// LS Electric XG5000 project: LOADER ITMV X3353 SYSTEM 20250323
// PLC LSPLC
// module base 0 slot 1: Internal Analog Input/Output:XBF-AH08E (A/D Voltage/Current 4 Ch, D/A Voltage/Current 4 Ch)
// module base 0 slot 2: Positioning Module:XBF-PN04B (Position Control, EtherCAT Network Type(4 axis))
// module base 0 slot 3: Input Module:XBE-DC32A (DC 24V Input, 32 Contacts (Current Source Sink Input/Current Source Input))

PROGRAM MAIN (task: ½ºÄµ ÇÁ·Î±×·¥)

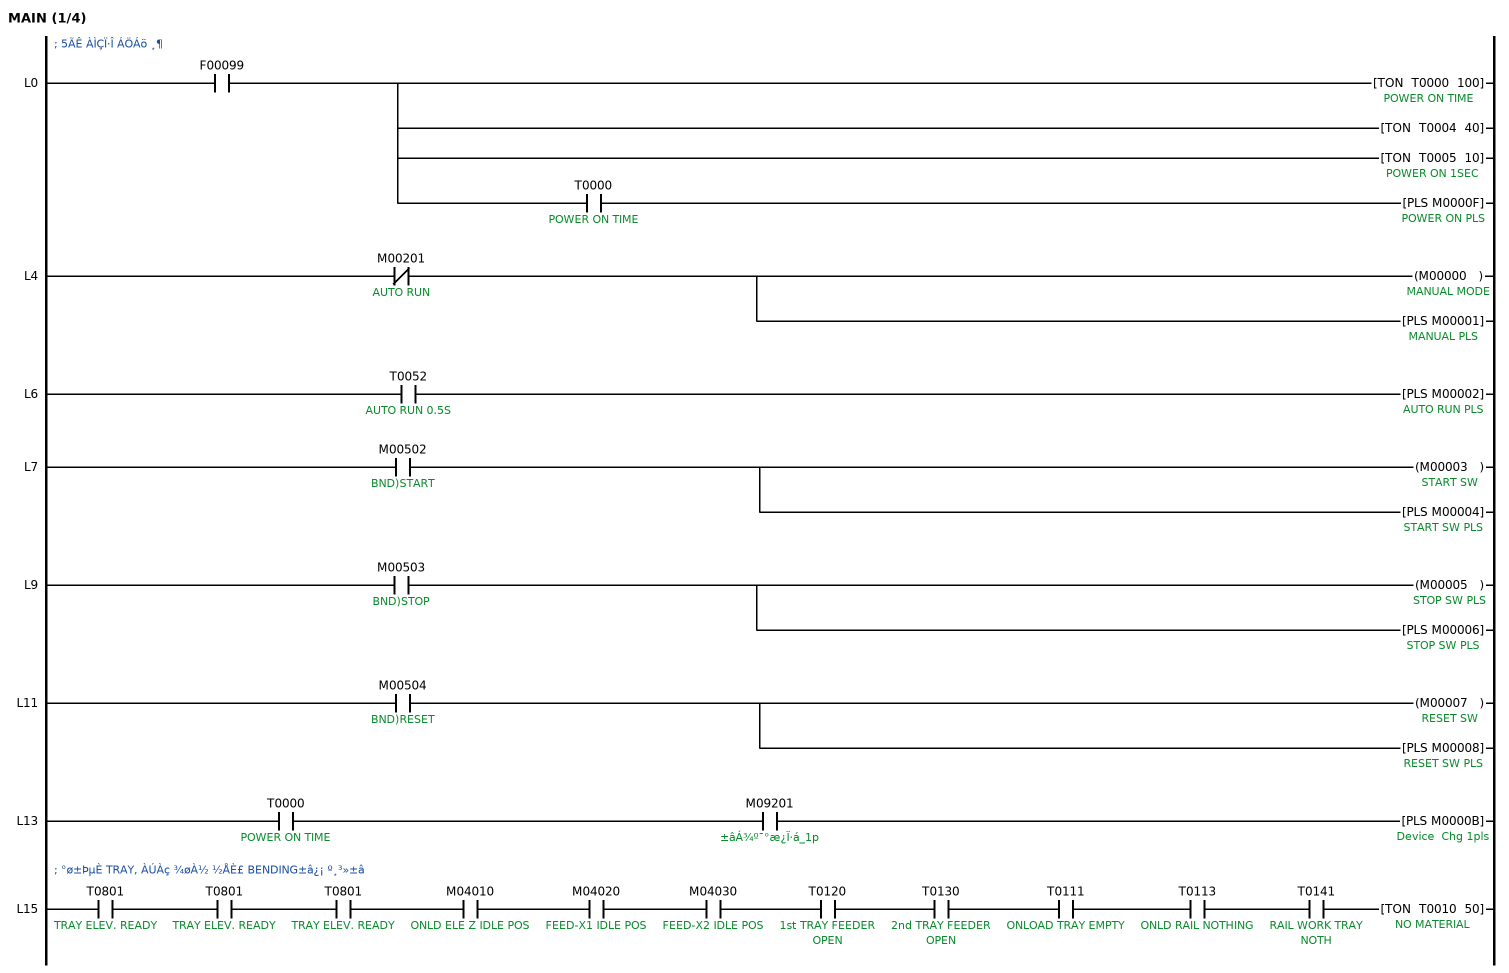
; L0
LOAD      F00099
TON       T0000 100	// POWER ON TIME
TON       T0004 40
TON       T0005 10	// POWER ON 1SEC
AND       T0000	// POWER ON TIME
OUTP      M0000F	// POWER ON PLS
// output comment: 5ÃÊ ÀÌÇÏ·Î ÁÖÁö ¸¶
; L4
LOAD NOT  M00201	// AUTO RUN
OUT       M00000	// MANUAL MODE
OUTP      M00001	// MANUAL PLS
; L6
LOAD      T0052	// AUTO RUN 0.5S
OUTP      M00002	// AUTO RUN PLS
; L7
LOAD      M00502	// BND)START
OUT       M00003	// START SW
OUTP      M00004	// START SW PLS
; L9
LOAD      M00503	// BND)STOP
OUT       M00005	// STOP SW PLS
OUTP      M00006	// STOP SW PLS
; L11
LOAD      M00504	// BND)RESET
OUT       M00007	// RESET SW
OUTP      M00008	// RESET SW PLS
; L13
LOAD      T0000	// POWER ON TIME
AND       M09201	// ±âÁ¾º¯°æ¿Ï·á_1p
OUTP      M0000B	// Device  Chg 1pls
// °ø±ÞµÈ TRAY, ÀÚÀç ¾øÀ½ ½ÅÈ£ BENDING±â¿¡ º¸³»±â
; L15
LOAD      T0801	// TRAY ELEV. READY
AND       T0801	// TRAY ELEV. READY
AND       T0801	// TRAY ELEV. READY
AND       M04010	// ONLD ELE Z IDLE POS
AND       M04020	// FEED-X1 IDLE POS
AND       M04030	// FEED-X2 IDLE POS
AND       T0120	// 1st TRAY FEEDER OPEN
AND       T0130	// 2nd TRAY FEEDER OPEN
AND       T0111	// ONLOAD TRAY EMPTY
AND       T0113	// ONLD RAIL NOTHING
AND       T0141	// RAIL WORK TRAY NOTH
TON       T0010 50	// NO MATERIAL

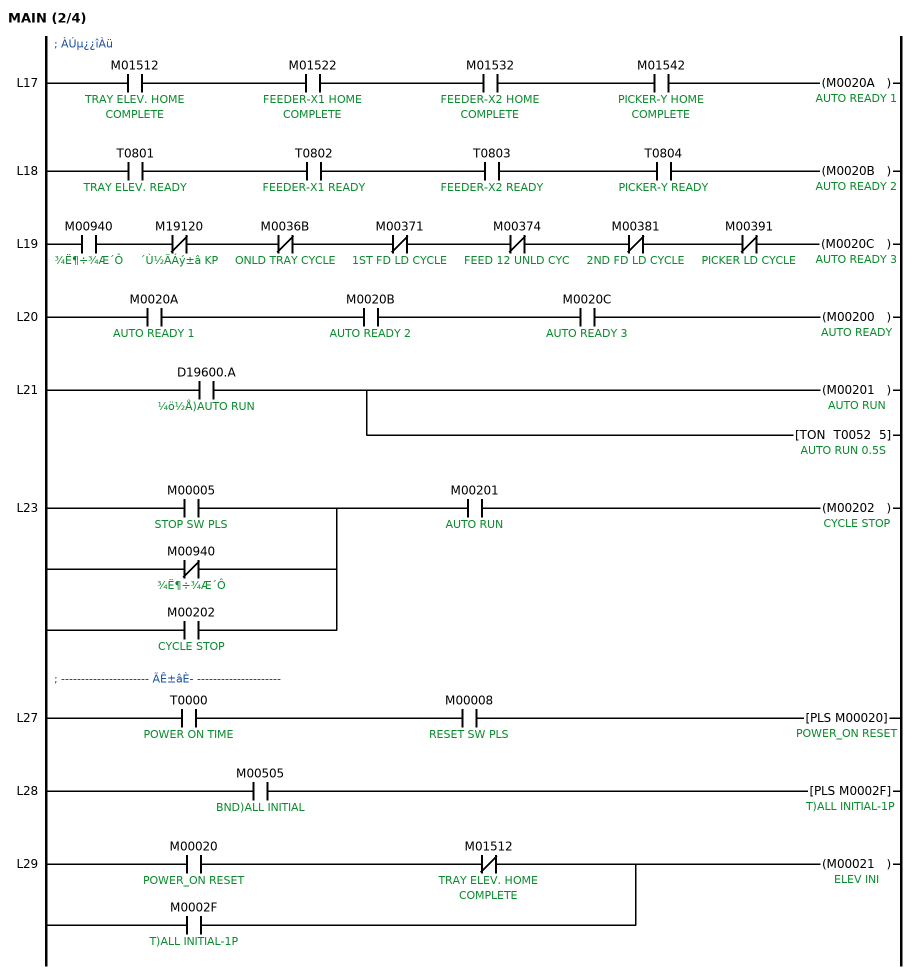
// ÀÚµ¿¿îÀü
; L17
LOAD      M01512	// TRAY ELEV. HOME COMPLETE
AND       M01522	// FEEDER-X1 HOME COMPLETE
AND       M01532	// FEEDER-X2 HOME COMPLETE
AND       M01542	// PICKER-Y HOME COMPLETE
OUT       M0020A	// AUTO READY 1
; L18
LOAD      T0801	// TRAY ELEV. READY
AND       T0802	// FEEDER-X1 READY
AND       T0803	// FEEDER-X2 READY
AND       T0804	// PICKER-Y READY
OUT       M0020B	// AUTO READY 2
; L19
LOAD      M00940	// ¾Ë¶÷¾Æ´Ô
AND NOT   M19120	// ´Ù½ÃÁý±â KP
AND NOT   M0036B	// ONLD TRAY CYCLE
AND NOT   M00371	// 1ST FD LD CYCLE
AND NOT   M00374	// FEED 12 UNLD CYC
AND NOT   M00381	// 2ND FD LD CYCLE
AND NOT   M00391	// PICKER LD CYCLE
OUT       M0020C	// AUTO READY 3
; L20
LOAD      M0020A	// AUTO READY 1
AND       M0020B	// AUTO READY 2
AND       M0020C	// AUTO READY 3
OUT       M00200	// AUTO READY
; L21
LOAD      D19600.A	// ¼ö½Å)AUTO RUN
OUT       M00201	// AUTO RUN
TON       T0052 5	// AUTO RUN 0.5S
; L23
LOAD      M00005	// STOP SW PLS
OR NOT    M00940	// ¾Ë¶÷¾Æ´Ô
OR        M00202	// CYCLE STOP
AND       M00201	// AUTO RUN
OUT       M00202	// CYCLE STOP
// ---------------------- ÃÊ±âÈ­ ---------------------
; L27
LOAD      T0000	// POWER ON TIME
AND       M00008	// RESET SW PLS
OUTP      M00020	// POWER_ON RESET
; L28
LOAD      M00505	// BND)ALL INITIAL
OUTP      M0002F	// T)ALL INITIAL-1P
; L29
LOAD      M00020	// POWER_ON RESET
AND NOT   M01512	// TRAY ELEV. HOME COMPLETE
OR        M0002F	// T)ALL INITIAL-1P
OUT       M00021	// ELEV INI

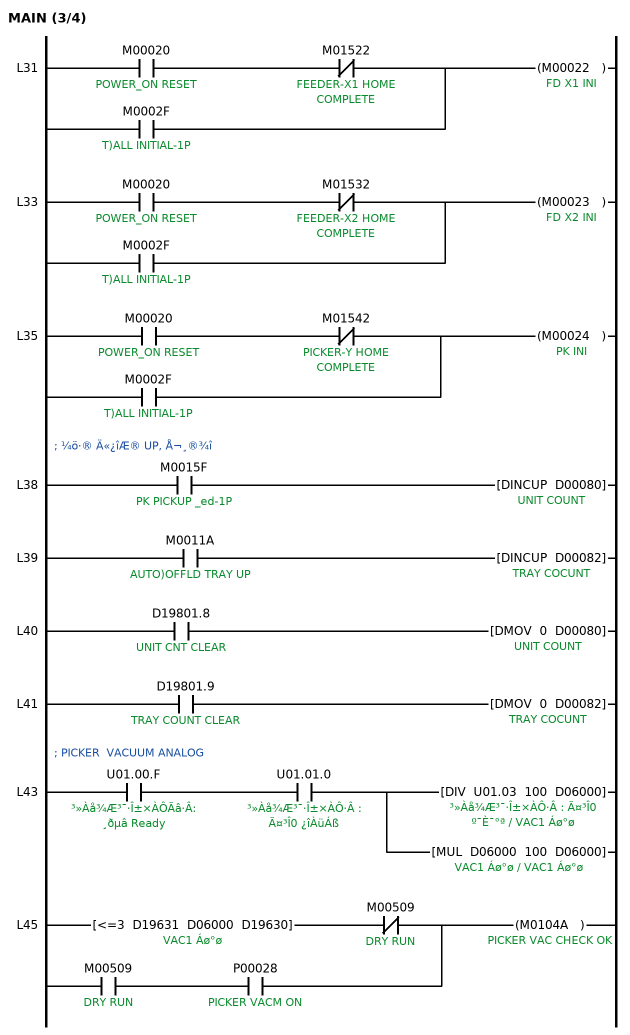
; L31
LOAD      M00020	// POWER_ON RESET
AND NOT   M01522	// FEEDER-X1 HOME COMPLETE
OR        M0002F	// T)ALL INITIAL-1P
OUT       M00022	// FD X1 INI
; L33
LOAD      M00020	// POWER_ON RESET
AND NOT   M01532	// FEEDER-X2 HOME COMPLETE
OR        M0002F	// T)ALL INITIAL-1P
OUT       M00023	// FD X2 INI
; L35
LOAD      M00020	// POWER_ON RESET
AND NOT   M01542	// PICKER-Y HOME COMPLETE
OR        M0002F	// T)ALL INITIAL-1P
OUT       M00024	// PK INI
// ¼ö·® Ä«¿îÆ® UP, Å¬¸®¾î
; L38
LOAD      M0015F	// PK PICKUP _ed-1P
DINCUP    D00080	// UNIT COUNT
; L39
LOAD      M0011A	// AUTO)OFFLD TRAY UP
DINCUP    D00082	// TRAY COCUNT
; L40
LOAD      D19801.8	// UNIT CNT CLEAR
DMOV      0 D00080	// UNIT COUNT
; L41
LOAD      D19801.9	// TRAY COUNT CLEAR
DMOV      0 D00082	// TRAY COCUNT
//   PICKER  VACUUM ANALOG
; L43
LOAD      U01.00.F	// ³»Àå¾Æ³¯·Î±×ÀÔÃâ·Â: ¸ðµâ Ready
AND       U01.01.0	// ³»Àå¾Æ³¯·Î±×ÀÔ·Â : Ã¤³Î0 ¿îÀüÁß
DIV       U01.03 100 D06000	// ³»Àå¾Æ³¯·Î±×ÀÔ·Â : Ã¤³Î0 º¯È¯°ª / VAC1 Áø°ø
MUL       D06000 100 D06000	// VAC1 Áø°ø / VAC1 Áø°ø
; L45
LOAD<=3   D19631 D06000 D19630	// VAC1 Áø°ø
AND NOT   M00509	// DRY RUN
LOAD      M00509	// DRY RUN
AND       P00028	// PICKER VACM ON
OR LOAD
OUT       M0104A	// PICKER VAC CHECK OK

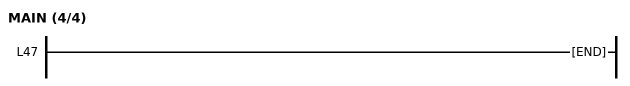
; L47
END

PROGRAM 01_ELEVATOR (task: ½ºÄµ ÇÁ·Î±×·¥)

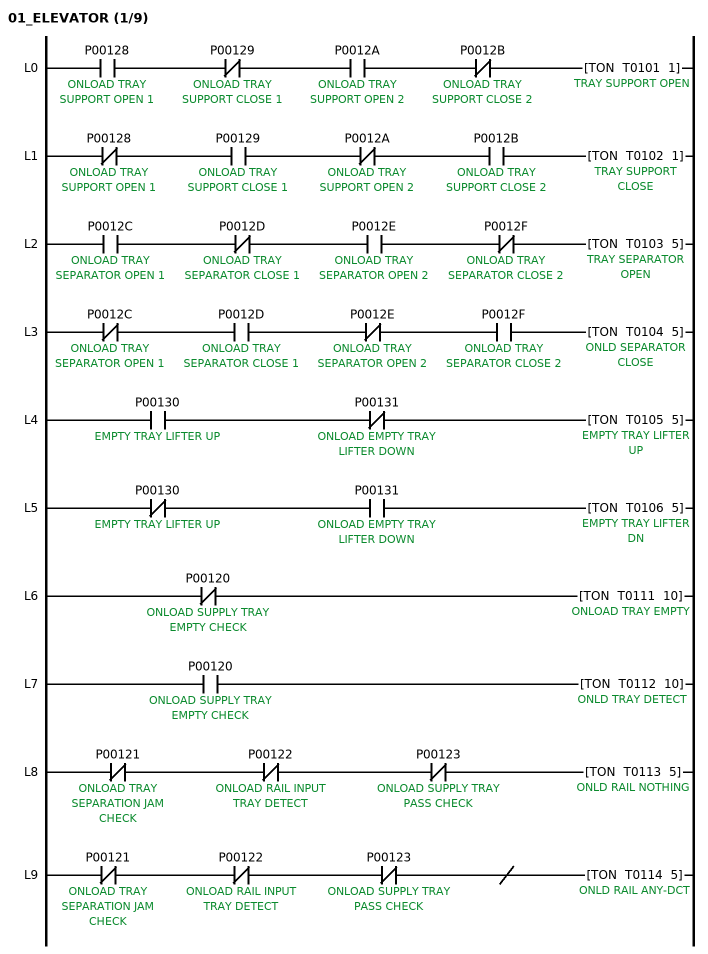
; L0
LOAD      P00128	// ONLOAD TRAY SUPPORT OPEN 1
AND NOT   P00129	// ONLOAD TRAY SUPPORT CLOSE 1
AND       P0012A	// ONLOAD TRAY SUPPORT OPEN 2
AND NOT   P0012B	// ONLOAD TRAY SUPPORT CLOSE 2
TON       T0101 1	// TRAY SUPPORT OPEN
; L1
LOAD NOT  P00128	// ONLOAD TRAY SUPPORT OPEN 1
AND       P00129	// ONLOAD TRAY SUPPORT CLOSE 1
AND NOT   P0012A	// ONLOAD TRAY SUPPORT OPEN 2
AND       P0012B	// ONLOAD TRAY SUPPORT CLOSE 2
TON       T0102 1	// TRAY SUPPORT CLOSE
; L2
LOAD      P0012C	// ONLOAD TRAY SEPARATOR OPEN 1
AND NOT   P0012D	// ONLOAD TRAY SEPARATOR CLOSE 1
AND       P0012E	// ONLOAD TRAY SEPARATOR OPEN 2
AND NOT   P0012F	// ONLOAD TRAY SEPARATOR CLOSE 2
TON       T0103 5	// TRAY SEPARATOR OPEN
; L3
LOAD NOT  P0012C	// ONLOAD TRAY SEPARATOR OPEN 1
AND       P0012D	// ONLOAD TRAY SEPARATOR CLOSE 1
AND NOT   P0012E	// ONLOAD TRAY SEPARATOR OPEN 2
AND       P0012F	// ONLOAD TRAY SEPARATOR CLOSE 2
TON       T0104 5	// ONLD SEPARATOR CLOSE
; L4
LOAD      P00130	// EMPTY TRAY LIFTER UP
AND NOT   P00131	// ONLOAD EMPTY TRAY LIFTER DOWN
TON       T0105 5	// EMPTY TRAY LIFTER UP
; L5
LOAD NOT  P00130	// EMPTY TRAY LIFTER UP
AND       P00131	// ONLOAD EMPTY TRAY LIFTER DOWN
TON       T0106 5	// EMPTY TRAY LIFTER DN
; L6
LOAD NOT  P00120	// ONLOAD SUPPLY TRAY EMPTY CHECK
TON       T0111 10	// ONLOAD TRAY EMPTY
; L7
LOAD      P00120	// ONLOAD SUPPLY TRAY EMPTY CHECK
TON       T0112 10	// ONLD TRAY DETECT
; L8
LOAD NOT  P00121	// ONLOAD TRAY SEPARATION JAM CHECK
AND NOT   P00122	// ONLOAD RAIL INPUT TRAY DETECT
AND NOT   P00123	// ONLOAD SUPPLY TRAY PASS CHECK
TON       T0113 5	// ONLD RAIL NOTHING
; L9
LOAD NOT  P00121	// ONLOAD TRAY SEPARATION JAM CHECK
AND NOT   P00122	// ONLOAD RAIL INPUT TRAY DETECT
AND NOT   P00123	// ONLOAD SUPPLY TRAY PASS CHECK
NOT
TON       T0114 5	// ONLD RAIL ANY-DCT

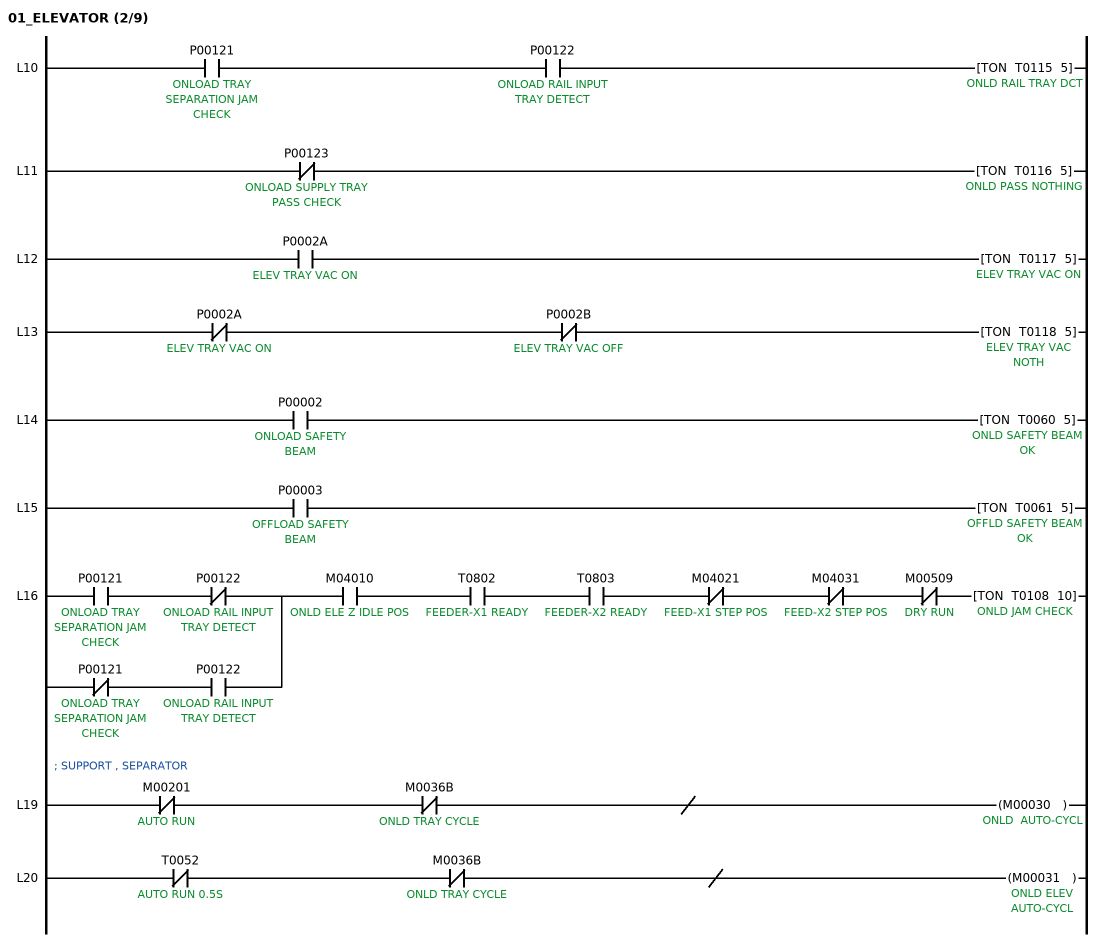
; L10
LOAD      P00121	// ONLOAD TRAY SEPARATION JAM CHECK
AND       P00122	// ONLOAD RAIL INPUT TRAY DETECT
TON       T0115 5	// ONLD RAIL TRAY DCT
; L11
LOAD NOT  P00123	// ONLOAD SUPPLY TRAY PASS CHECK
TON       T0116 5	// ONLD PASS NOTHING
; L12
LOAD      P0002A	// ELEV TRAY VAC ON
TON       T0117 5	// ELEV TRAY VAC ON
; L13
LOAD NOT  P0002A	// ELEV TRAY VAC ON
AND NOT   P0002B	// ELEV TRAY VAC OFF
TON       T0118 5	// ELEV TRAY VAC NOTH
; L14
LOAD      P00002	// ONLOAD SAFETY BEAM
TON       T0060 5	// ONLD SAFETY BEAM OK
; L15
LOAD      P00003	// OFFLOAD SAFETY BEAM
TON       T0061 5	// OFFLD SAFETY BEAM OK
; L16
LOAD      P00121	// ONLOAD TRAY SEPARATION JAM CHECK
AND NOT   P00122	// ONLOAD RAIL INPUT TRAY DETECT
LOAD NOT  P00121	// ONLOAD TRAY SEPARATION JAM CHECK
AND       P00122	// ONLOAD RAIL INPUT TRAY DETECT
OR LOAD
AND       M04010	// ONLD ELE Z IDLE POS
AND       T0802	// FEEDER-X1 READY
AND       T0803	// FEEDER-X2 READY
AND NOT   M04021	// FEED-X1 STEP POS
AND NOT   M04031	// FEED-X2 STEP POS
AND NOT   M00509	// DRY RUN
TON       T0108 10	// ONLD JAM CHECK
// SUPPORT , SEPARATOR
; L19
LOAD NOT  M00201	// AUTO RUN
AND NOT   M0036B	// ONLD TRAY CYCLE
NOT
OUT       M00030	// ONLD  AUTO-CYCL
; L20
LOAD NOT  T0052	// AUTO RUN 0.5S
AND NOT   M0036B	// ONLD TRAY CYCLE
NOT
OUT       M00031	// ONLD ELEV AUTO-CYCL

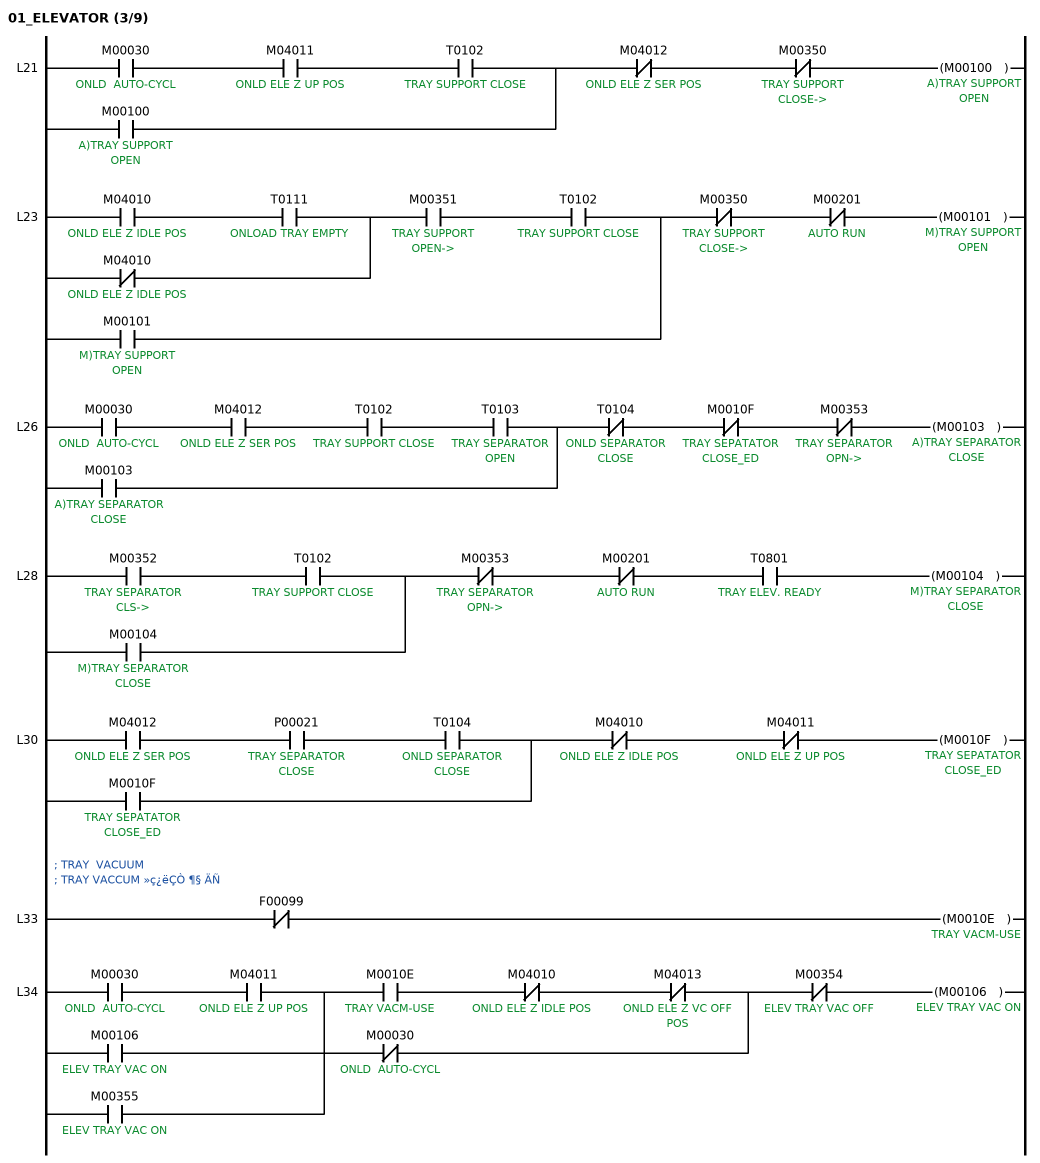
; L21
LOAD      M00030	// ONLD  AUTO-CYCL
AND       M04011	// ONLD ELE Z UP POS
AND       T0102	// TRAY SUPPORT CLOSE
OR        M00100	// A)TRAY SUPPORT OPEN
AND NOT   M04012	// ONLD ELE Z SER POS
AND NOT   M00350	// TRAY SUPPORT CLOSE->
OUT       M00100	// A)TRAY SUPPORT OPEN
; L23
LOAD      M04010	// ONLD ELE Z IDLE POS
AND       T0111	// ONLOAD TRAY EMPTY
OR NOT    M04010	// ONLD ELE Z IDLE POS
AND       M00351	// TRAY SUPPORT OPEN->
AND       T0102	// TRAY SUPPORT CLOSE
OR        M00101	// M)TRAY SUPPORT OPEN
AND NOT   M00350	// TRAY SUPPORT CLOSE->
AND NOT   M00201	// AUTO RUN
OUT       M00101	// M)TRAY SUPPORT OPEN
; L26
LOAD      M00030	// ONLD  AUTO-CYCL
AND       M04012	// ONLD ELE Z SER POS
AND       T0102	// TRAY SUPPORT CLOSE
AND       T0103	// TRAY SEPARATOR OPEN
OR        M00103	// A)TRAY SEPARATOR CLOSE
AND NOT   T0104	// ONLD SEPARATOR CLOSE
AND NOT   M0010F	// TRAY SEPATATOR CLOSE_ED
AND NOT   M00353	// TRAY SEPARATOR OPN->
OUT       M00103	// A)TRAY SEPARATOR CLOSE
; L28
LOAD      M00352	// TRAY SEPARATOR CLS->
AND       T0102	// TRAY SUPPORT CLOSE
OR        M00104	// M)TRAY SEPARATOR CLOSE
AND NOT   M00353	// TRAY SEPARATOR OPN->
AND NOT   M00201	// AUTO RUN
AND       T0801	// TRAY ELEV. READY
OUT       M00104	// M)TRAY SEPARATOR CLOSE
; L30
LOAD      M04012	// ONLD ELE Z SER POS
AND       P00021	// TRAY SEPARATOR CLOSE
AND       T0104	// ONLD SEPARATOR CLOSE
OR        M0010F	// TRAY SEPATATOR CLOSE_ED
AND NOT   M04010	// ONLD ELE Z IDLE POS
AND NOT   M04011	// ONLD ELE Z UP POS
OUT       M0010F	// TRAY SEPATATOR CLOSE_ED
// TRAY  VACUUM
; L33
LOAD NOT  F00099
OUT       M0010E	// TRAY VACM-USE
// output comment: TRAY VACCUM »ç¿ëÇÒ ¶§ ÄÑ
; L34
LOAD      M00030	// ONLD  AUTO-CYCL
AND       M04011	// ONLD ELE Z UP POS
OR        M00106	// ELEV TRAY VAC ON
OR        M00355	// ELEV TRAY VAC ON
LOAD      M0010E	// TRAY VACM-USE
AND NOT   M04010	// ONLD ELE Z IDLE POS
AND NOT   M04013	// ONLD ELE Z VC OFF POS
OR NOT    M00030	// ONLD  AUTO-CYCL
AND LOAD
AND NOT   M00354	// ELEV TRAY VAC OFF
OUT       M00106	// ELEV TRAY VAC ON

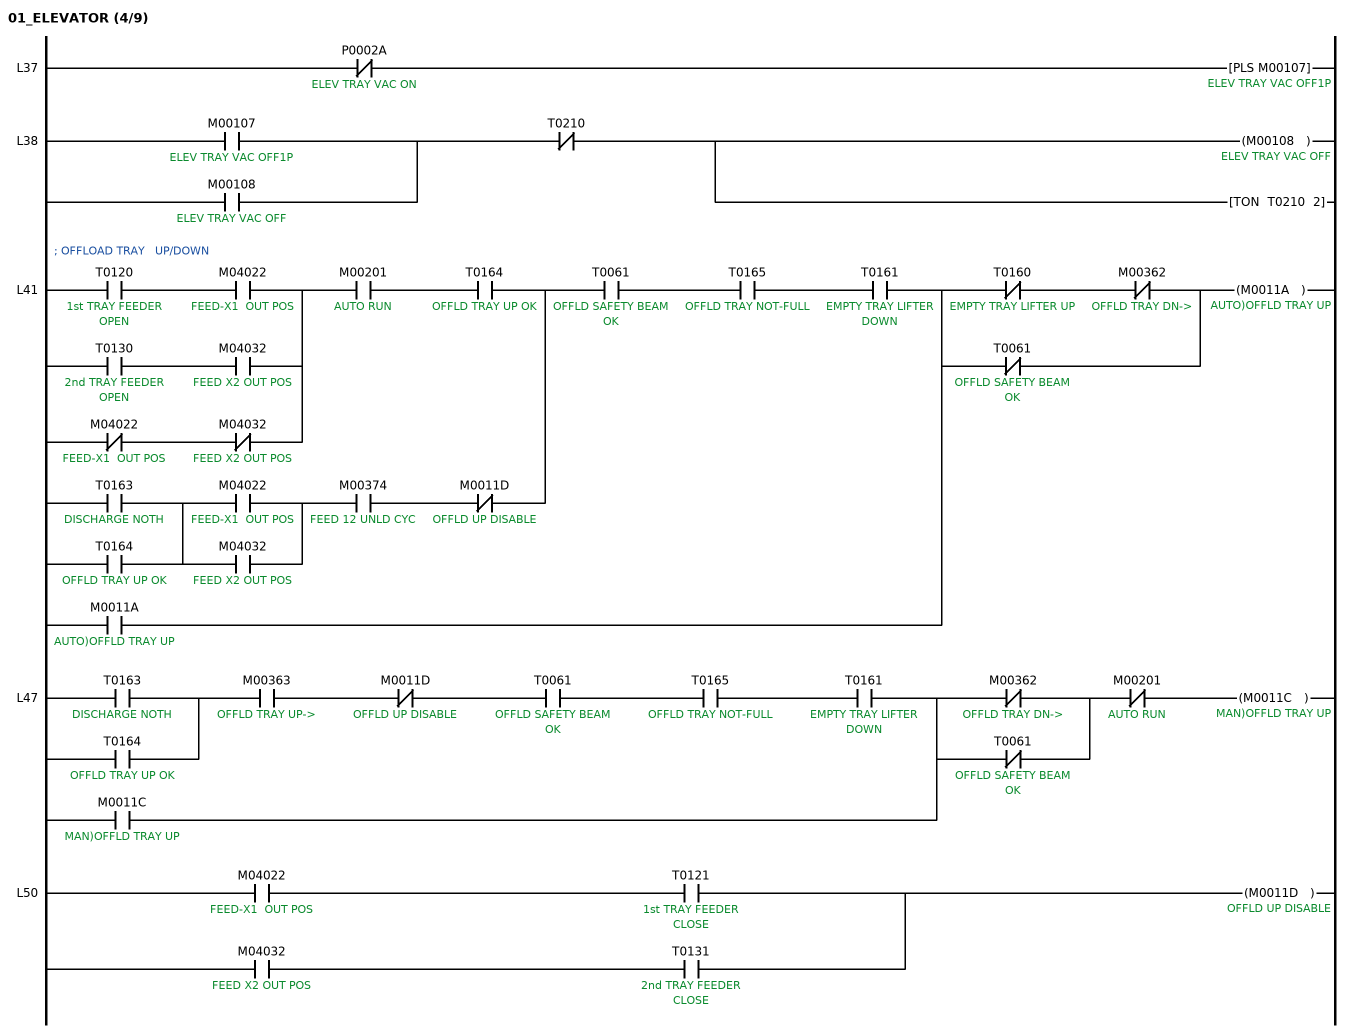
; L37
LOAD NOT  P0002A	// ELEV TRAY VAC ON
OUTP      M00107	// ELEV TRAY VAC OFF1P
; L38
LOAD      M00107	// ELEV TRAY VAC OFF1P
OR        M00108	// ELEV TRAY VAC OFF
AND NOT   T0210
OUT       M00108	// ELEV TRAY VAC OFF
TON       T0210 2
// OFFLOAD TRAY   UP/DOWN
; L41
LOAD      T0120	// 1st TRAY FEEDER OPEN
AND       M04022	// FEED-X1  OUT POS
LOAD      T0130	// 2nd TRAY FEEDER OPEN
AND       M04032	// FEED X2 OUT POS
OR LOAD
LOAD NOT  M04022	// FEED-X1  OUT POS
AND NOT   M04032	// FEED X2 OUT POS
OR LOAD
AND       M00201	// AUTO RUN
AND       T0164	// OFFLD TRAY UP OK
LOAD      T0163	// DISCHARGE NOTH
OR        T0164	// OFFLD TRAY UP OK
LOAD      M04022	// FEED-X1  OUT POS
OR        M04032	// FEED X2 OUT POS
AND LOAD
AND       M00374	// FEED 12 UNLD CYC
AND NOT   M0011D	// OFFLD UP DISABLE
OR LOAD
AND       T0061	// OFFLD SAFETY BEAM OK
AND       T0165	// OFFLD TRAY NOT-FULL
AND       T0161	// EMPTY TRAY LIFTER DOWN
OR        M0011A	// AUTO)OFFLD TRAY UP
LOAD NOT  T0160	// EMPTY TRAY LIFTER UP
AND NOT   M00362	// OFFLD TRAY DN->
OR NOT    T0061	// OFFLD SAFETY BEAM OK
AND LOAD
OUT       M0011A	// AUTO)OFFLD TRAY UP
; L47
LOAD      T0163	// DISCHARGE NOTH
OR        T0164	// OFFLD TRAY UP OK
AND       M00363	// OFFLD TRAY UP->
AND NOT   M0011D	// OFFLD UP DISABLE
AND       T0061	// OFFLD SAFETY BEAM OK
AND       T0165	// OFFLD TRAY NOT-FULL
AND       T0161	// EMPTY TRAY LIFTER DOWN
OR        M0011C	// MAN)OFFLD TRAY UP
LOAD NOT  M00362	// OFFLD TRAY DN->
OR NOT    T0061	// OFFLD SAFETY BEAM OK
AND LOAD
AND NOT   M00201	// AUTO RUN
OUT       M0011C	// MAN)OFFLD TRAY UP
; L50
LOAD      M04022	// FEED-X1  OUT POS
AND       T0121	// 1st TRAY FEEDER CLOSE
LOAD      M04032	// FEED X2 OUT POS
AND       T0131	// 2nd TRAY FEEDER CLOSE
OR LOAD
OUT       M0011D	// OFFLD UP DISABLE

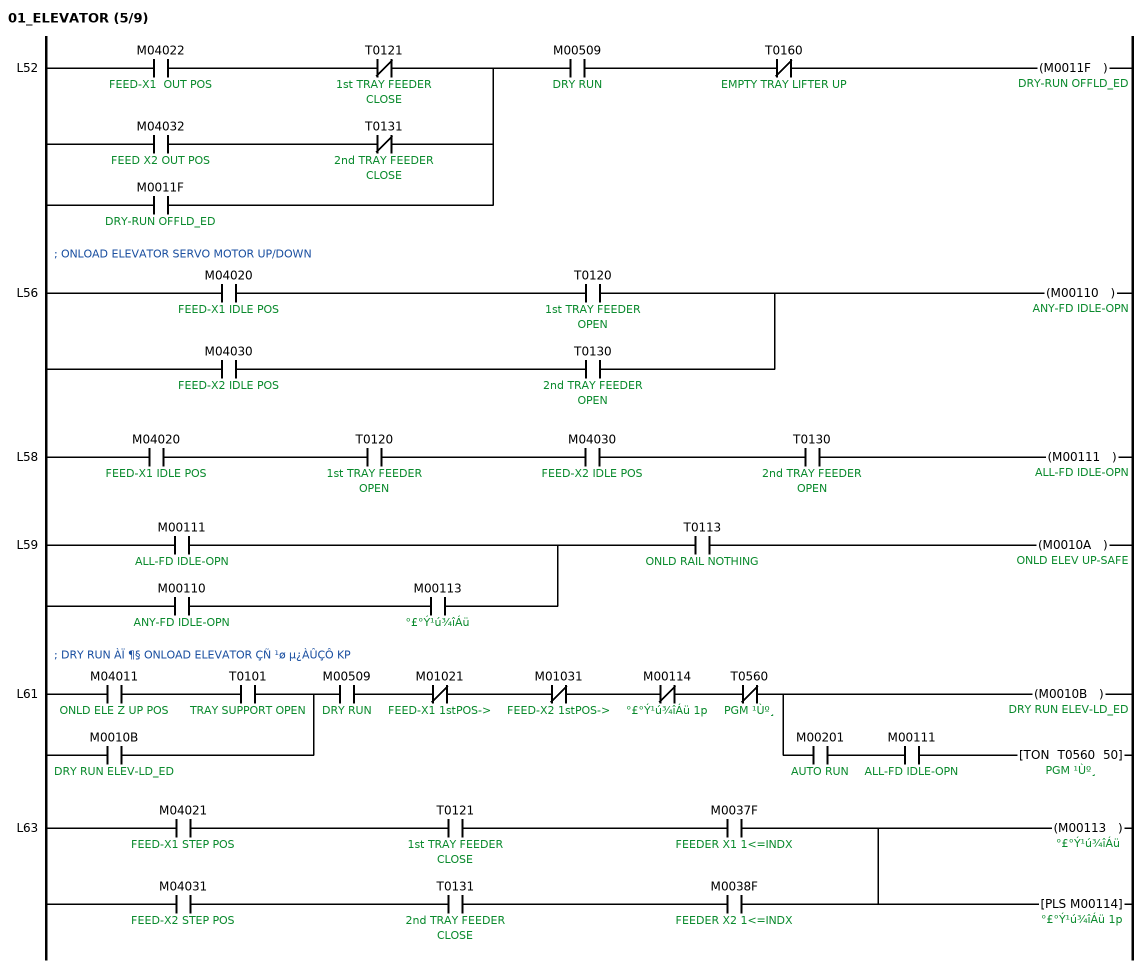
; L52
LOAD      M04022	// FEED-X1  OUT POS
AND NOT   T0121	// 1st TRAY FEEDER CLOSE
LOAD      M04032	// FEED X2 OUT POS
AND NOT   T0131	// 2nd TRAY FEEDER CLOSE
OR LOAD
OR        M0011F	// DRY-RUN OFFLD_ED
AND       M00509	// DRY RUN
AND NOT   T0160	// EMPTY TRAY LIFTER UP
OUT       M0011F	// DRY-RUN OFFLD_ED
// ONLOAD ELEVATOR SERVO MOTOR UP/DOWN
; L56
LOAD      M04020	// FEED-X1 IDLE POS
AND       T0120	// 1st TRAY FEEDER OPEN
LOAD      M04030	// FEED-X2 IDLE POS
AND       T0130	// 2nd TRAY FEEDER OPEN
OR LOAD
OUT       M00110	// ANY-FD IDLE-OPN
; L58
LOAD      M04020	// FEED-X1 IDLE POS
AND       T0120	// 1st TRAY FEEDER OPEN
AND       M04030	// FEED-X2 IDLE POS
AND       T0130	// 2nd TRAY FEEDER OPEN
OUT       M00111	// ALL-FD IDLE-OPN
; L59
LOAD      M00111	// ALL-FD IDLE-OPN
LOAD      M00110	// ANY-FD IDLE-OPN
AND       M00113	// °£°Ý¹ú¾îÁü
OR LOAD
AND       T0113	// ONLD RAIL NOTHING
OUT       M0010A	// ONLD ELEV UP-SAFE
; L61
LOAD      M04011	// ONLD ELE Z UP POS
AND       T0101	// TRAY SUPPORT OPEN
OR        M0010B	// DRY RUN ELEV-LD_ED
AND       M00509	// DRY RUN
AND NOT   M01021	// FEED-X1 1stPOS->
AND NOT   M01031	// FEED-X2 1stPOS->
AND NOT   M00114	// °£°Ý¹ú¾îÁü 1p
AND NOT   T0560	// PGM ¹Ùº¸
OUT       M0010B	// DRY RUN ELEV-LD_ED
AND       M00201	// AUTO RUN
AND       M00111	// ALL-FD IDLE-OPN
TON       T0560 50	// PGM ¹Ùº¸
// output comment: DRY RUN ÀÏ ¶§ ONLOAD ELEVATOR ÇÑ ¹ø µ¿ÀÛÇÔ KP
; L63
LOAD      M04021	// FEED-X1 STEP POS
AND       T0121	// 1st TRAY FEEDER CLOSE
AND       M0037F	// FEEDER X1 1<=INDX
LOAD      M04031	// FEED-X2 STEP POS
AND       T0131	// 2nd TRAY FEEDER CLOSE
AND       M0038F	// FEEDER X2 1<=INDX
OR LOAD
OUT       M00113	// °£°Ý¹ú¾îÁü
OUTP      M00114	// °£°Ý¹ú¾îÁü 1p

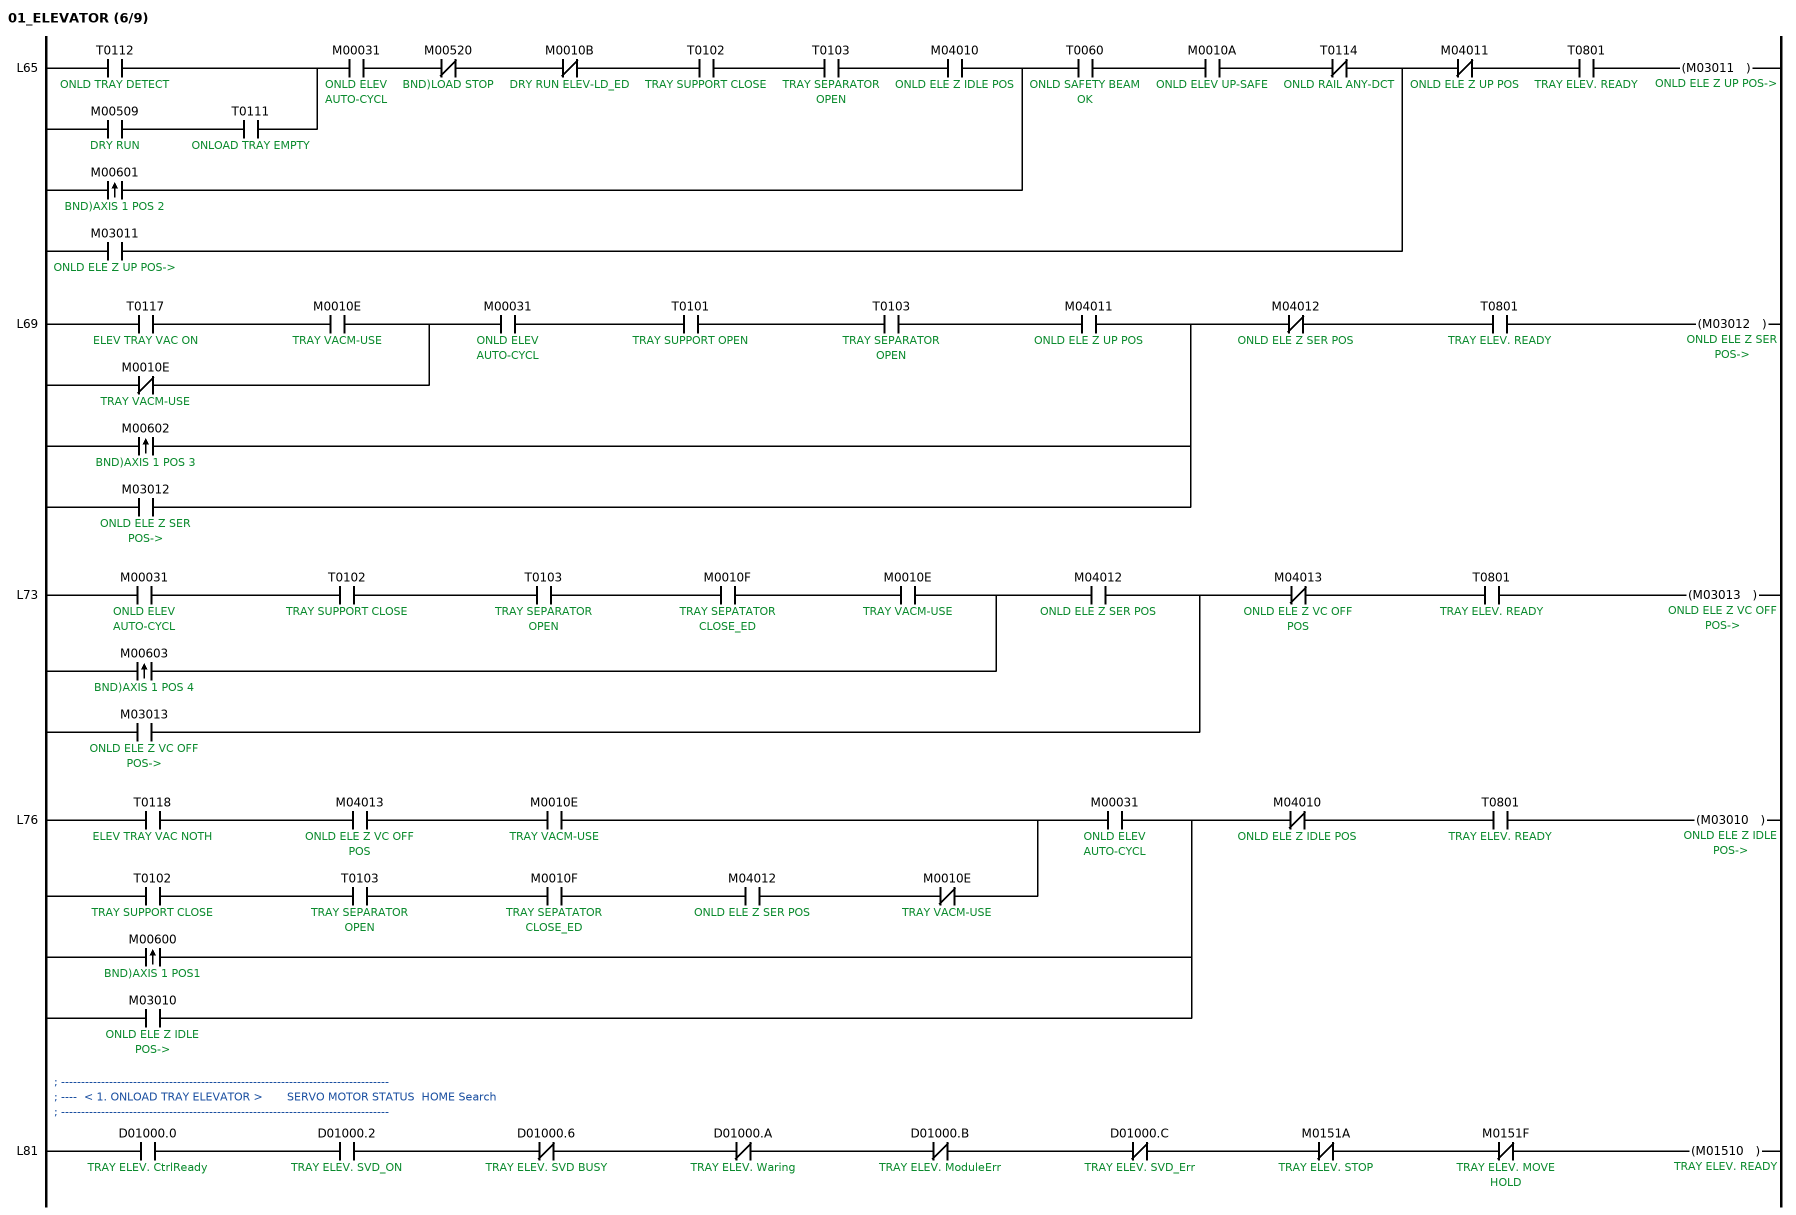
; L65
LOAD      T0112	// ONLD TRAY DETECT
LOAD      M00509	// DRY RUN
AND       T0111	// ONLOAD TRAY EMPTY
OR LOAD
AND       M00031	// ONLD ELEV AUTO-CYCL
AND NOT   M00520	// BND)LOAD STOP
AND NOT   M0010B	// DRY RUN ELEV-LD_ED
AND       T0102	// TRAY SUPPORT CLOSE
AND       T0103	// TRAY SEPARATOR OPEN
AND       M04010	// ONLD ELE Z IDLE POS
ORP       M00601	// BND)AXIS 1 POS 2
AND       T0060	// ONLD SAFETY BEAM OK
AND       M0010A	// ONLD ELEV UP-SAFE
AND NOT   T0114	// ONLD RAIL ANY-DCT
OR        M03011	// ONLD ELE Z UP POS->
AND NOT   M04011	// ONLD ELE Z UP POS
AND       T0801	// TRAY ELEV. READY
OUT       M03011	// ONLD ELE Z UP POS->
; L69
LOAD      T0117	// ELEV TRAY VAC ON
AND       M0010E	// TRAY VACM-USE
OR NOT    M0010E	// TRAY VACM-USE
AND       M00031	// ONLD ELEV AUTO-CYCL
AND       T0101	// TRAY SUPPORT OPEN
AND       T0103	// TRAY SEPARATOR OPEN
AND       M04011	// ONLD ELE Z UP POS
ORP       M00602	// BND)AXIS 1 POS 3
OR        M03012	// ONLD ELE Z SER POS->
AND NOT   M04012	// ONLD ELE Z SER POS
AND       T0801	// TRAY ELEV. READY
OUT       M03012	// ONLD ELE Z SER POS->
; L73
LOAD      M00031	// ONLD ELEV AUTO-CYCL
AND       T0102	// TRAY SUPPORT CLOSE
AND       T0103	// TRAY SEPARATOR OPEN
AND       M0010F	// TRAY SEPATATOR CLOSE_ED
AND       M0010E	// TRAY VACM-USE
ORP       M00603	// BND)AXIS 1 POS 4
AND       M04012	// ONLD ELE Z SER POS
OR        M03013	// ONLD ELE Z VC OFF POS->
AND NOT   M04013	// ONLD ELE Z VC OFF POS
AND       T0801	// TRAY ELEV. READY
OUT       M03013	// ONLD ELE Z VC OFF POS->
; L76
LOAD      T0118	// ELEV TRAY VAC NOTH
AND       M04013	// ONLD ELE Z VC OFF POS
AND       M0010E	// TRAY VACM-USE
LOAD      T0102	// TRAY SUPPORT CLOSE
AND       T0103	// TRAY SEPARATOR OPEN
AND       M0010F	// TRAY SEPATATOR CLOSE_ED
AND       M04012	// ONLD ELE Z SER POS
AND NOT   M0010E	// TRAY VACM-USE
OR LOAD
AND       M00031	// ONLD ELEV AUTO-CYCL
ORP       M00600	// BND)AXIS 1 POS1
OR        M03010	// ONLD ELE Z IDLE POS->
AND NOT   M04010	// ONLD ELE Z IDLE POS
AND       T0801	// TRAY ELEV. READY
OUT       M03010	// ONLD ELE Z IDLE POS->
// ----------------------------------------------------------------------------------
// 
// ----  < 1. ONLOAD TRAY ELEVATOR >       SERVO MOTOR STATUS  HOME Search
// 
// ----------------------------------------------------------------------------------
; L81
LOAD      D01000.0	// TRAY ELEV. CtrlReady
AND       D01000.2	// TRAY ELEV. SVD_ON
AND NOT   D01000.6	// TRAY ELEV. SVD BUSY
AND NOT   D01000.A	// TRAY ELEV. Waring
AND NOT   D01000.B	// TRAY ELEV. ModuleErr
AND NOT   D01000.C	// TRAY ELEV. SVD_Err
AND NOT   M0151A	// TRAY ELEV. STOP
AND NOT   M0151F	// TRAY ELEV. MOVE HOLD
OUT       M01510	// TRAY ELEV. READY

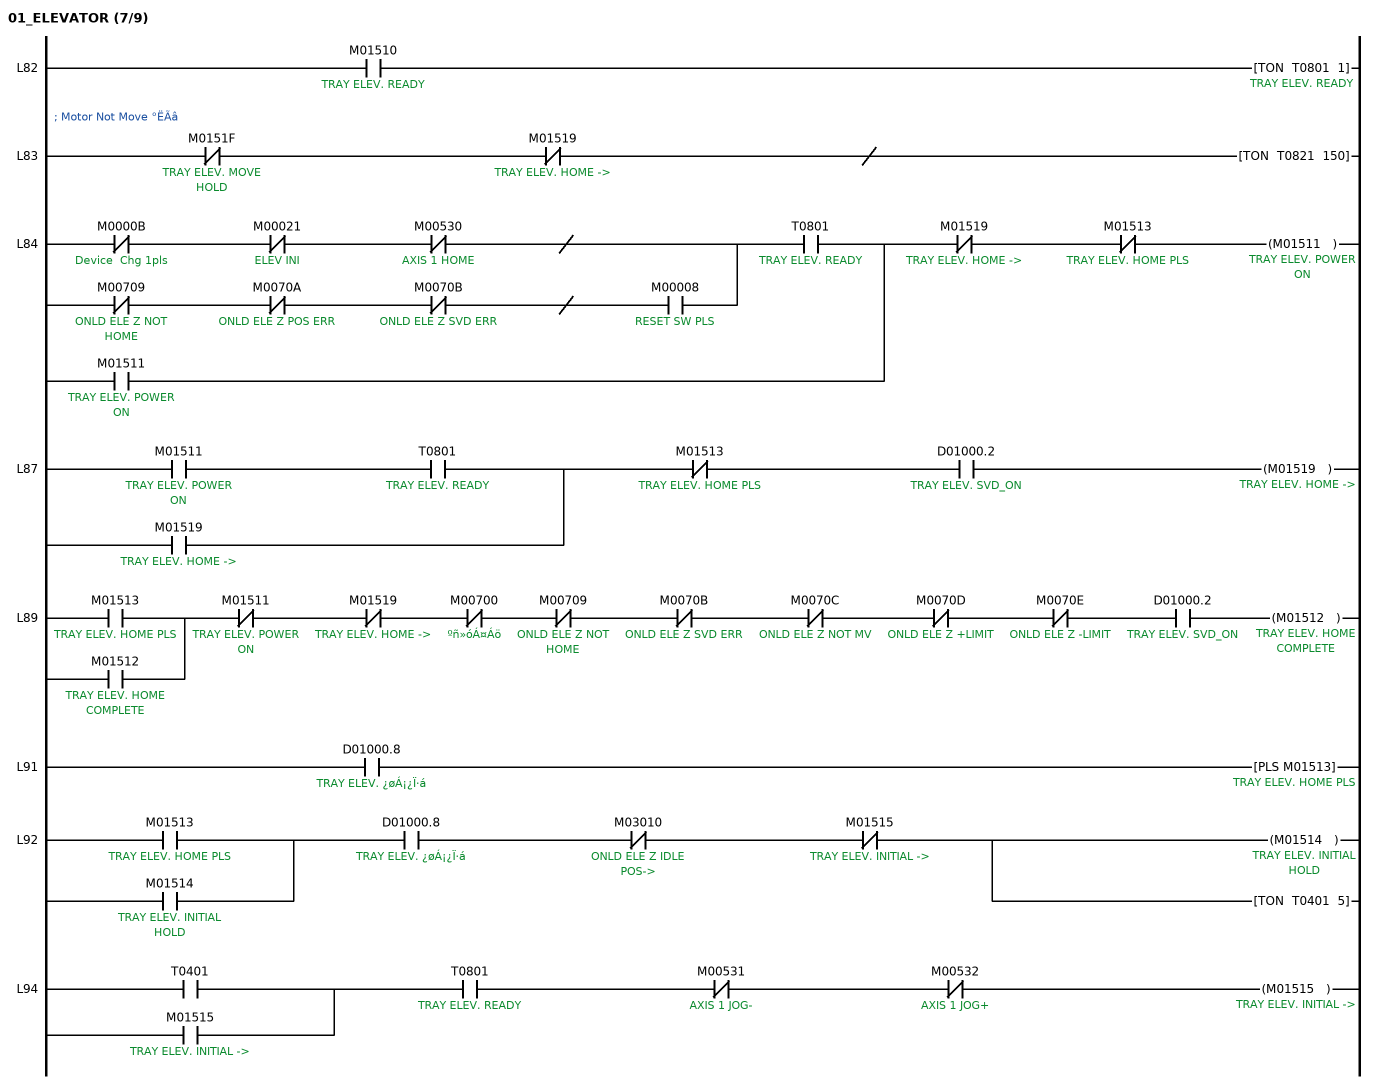
; L82
LOAD      M01510	// TRAY ELEV. READY
TON       T0801 1	// TRAY ELEV. READY
; L83
LOAD NOT  M0151F	// TRAY ELEV. MOVE HOLD
AND NOT   M01519	// TRAY ELEV. HOME ->
NOT
TON       T0821 150
// output comment: Motor Not Move °ËÃâ
; L84
LOAD NOT  M0000B	// Device  Chg 1pls
AND NOT   M00021	// ELEV INI
AND NOT   M00530	// AXIS 1 HOME
NOT
LOAD NOT  M00709	// ONLD ELE Z NOT HOME
AND NOT   M0070A	// ONLD ELE Z POS ERR
AND NOT   M0070B	// ONLD ELE Z SVD ERR
NOT
AND       M00008	// RESET SW PLS
OR LOAD
AND       T0801	// TRAY ELEV. READY
OR        M01511	// TRAY ELEV. POWER ON
AND NOT   M01519	// TRAY ELEV. HOME ->
AND NOT   M01513	// TRAY ELEV. HOME PLS
OUT       M01511	// TRAY ELEV. POWER ON
; L87
LOAD      M01511	// TRAY ELEV. POWER ON
AND       T0801	// TRAY ELEV. READY
OR        M01519	// TRAY ELEV. HOME ->
AND NOT   M01513	// TRAY ELEV. HOME PLS
AND       D01000.2	// TRAY ELEV. SVD_ON
OUT       M01519	// TRAY ELEV. HOME ->
; L89
LOAD      M01513	// TRAY ELEV. HOME PLS
OR        M01512	// TRAY ELEV. HOME COMPLETE
AND NOT   M01511	// TRAY ELEV. POWER ON
AND NOT   M01519	// TRAY ELEV. HOME ->
AND NOT   M00700	// ºñ»óÁ¤Áö
AND NOT   M00709	// ONLD ELE Z NOT HOME
AND NOT   M0070B	// ONLD ELE Z SVD ERR
AND NOT   M0070C	// ONLD ELE Z NOT MV
AND NOT   M0070D	// ONLD ELE Z +LIMIT
AND NOT   M0070E	// ONLD ELE Z -LIMIT
AND       D01000.2	// TRAY ELEV. SVD_ON
OUT       M01512	// TRAY ELEV. HOME COMPLETE
; L91
LOAD      D01000.8	// TRAY ELEV. ¿øÁ¡¿Ï·á
OUTP      M01513	// TRAY ELEV. HOME PLS
; L92
LOAD      M01513	// TRAY ELEV. HOME PLS
OR        M01514	// TRAY ELEV. INITIAL HOLD
AND       D01000.8	// TRAY ELEV. ¿øÁ¡¿Ï·á
AND NOT   M03010	// ONLD ELE Z IDLE POS->
AND NOT   M01515	// TRAY ELEV. INITIAL ->
OUT       M01514	// TRAY ELEV. INITIAL HOLD
TON       T0401 5
; L94
LOAD      T0401
OR        M01515	// TRAY ELEV. INITIAL ->
AND       T0801	// TRAY ELEV. READY
AND NOT   M00531	// AXIS 1 JOG-
AND NOT   M00532	// AXIS 1 JOG+
OUT       M01515	// TRAY ELEV. INITIAL ->

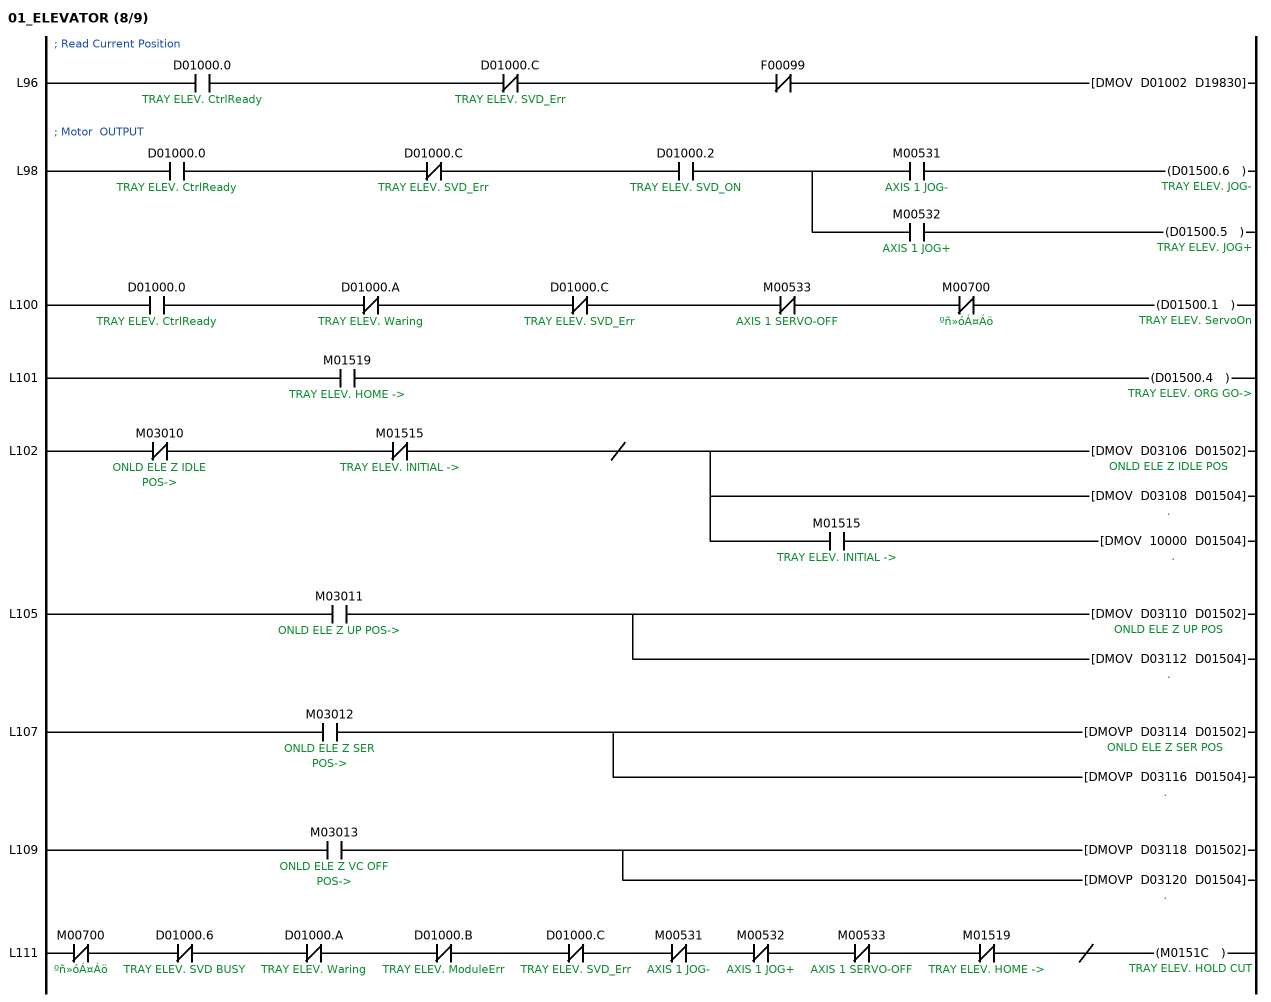
; L96
LOAD      D01000.0	// TRAY ELEV. CtrlReady
AND NOT   D01000.C	// TRAY ELEV. SVD_Err
AND NOT   F00099
DMOV      D01002 D19830
// output comment: Read Current Position
//  Motor  OUTPUT
; L98
LOAD      D01000.0	// TRAY ELEV. CtrlReady
AND NOT   D01000.C	// TRAY ELEV. SVD_Err
AND       D01000.2	// TRAY ELEV. SVD_ON
MPUSH
AND       M00531	// AXIS 1 JOG-
OUT       D01500.6	// TRAY ELEV. JOG-
MPOP
AND       M00532	// AXIS 1 JOG+
OUT       D01500.5	// TRAY ELEV. JOG+
; L100
LOAD      D01000.0	// TRAY ELEV. CtrlReady
AND NOT   D01000.A	// TRAY ELEV. Waring
AND NOT   D01000.C	// TRAY ELEV. SVD_Err
AND NOT   M00533	// AXIS 1 SERVO-OFF
AND NOT   M00700	// ºñ»óÁ¤Áö
OUT       D01500.1	// TRAY ELEV. ServoOn
; L101
LOAD      M01519	// TRAY ELEV. HOME ->
OUT       D01500.4	// TRAY ELEV. ORG GO->
; L102
LOAD NOT  M03010	// ONLD ELE Z IDLE POS->
AND NOT   M01515	// TRAY ELEV. INITIAL ->
NOT
DMOV      D03106 D01502	// ONLD ELE Z IDLE POS
DMOV      D03108 D01504	// .
AND       M01515	// TRAY ELEV. INITIAL ->
DMOV      10000 D01504	// .
; L105
LOAD      M03011	// ONLD ELE Z UP POS->
DMOV      D03110 D01502	// ONLD ELE Z UP POS
DMOV      D03112 D01504	// .
; L107
LOAD      M03012	// ONLD ELE Z SER POS->
DMOVP     D03114 D01502	// ONLD ELE Z SER POS
DMOVP     D03116 D01504	// .
; L109
LOAD      M03013	// ONLD ELE Z VC OFF POS->
DMOVP     D03118 D01502
DMOVP     D03120 D01504	// .
; L111
LOAD NOT  M00700	// ºñ»óÁ¤Áö
AND NOT   D01000.6	// TRAY ELEV. SVD BUSY
AND NOT   D01000.A	// TRAY ELEV. Waring
AND NOT   D01000.B	// TRAY ELEV. ModuleErr
AND NOT   D01000.C	// TRAY ELEV. SVD_Err
AND NOT   M00531	// AXIS 1 JOG-
AND NOT   M00532	// AXIS 1 JOG+
AND NOT   M00533	// AXIS 1 SERVO-OFF
AND NOT   M01519	// TRAY ELEV. HOME ->
NOT
OUT       M0151C	// TRAY ELEV. HOLD CUT

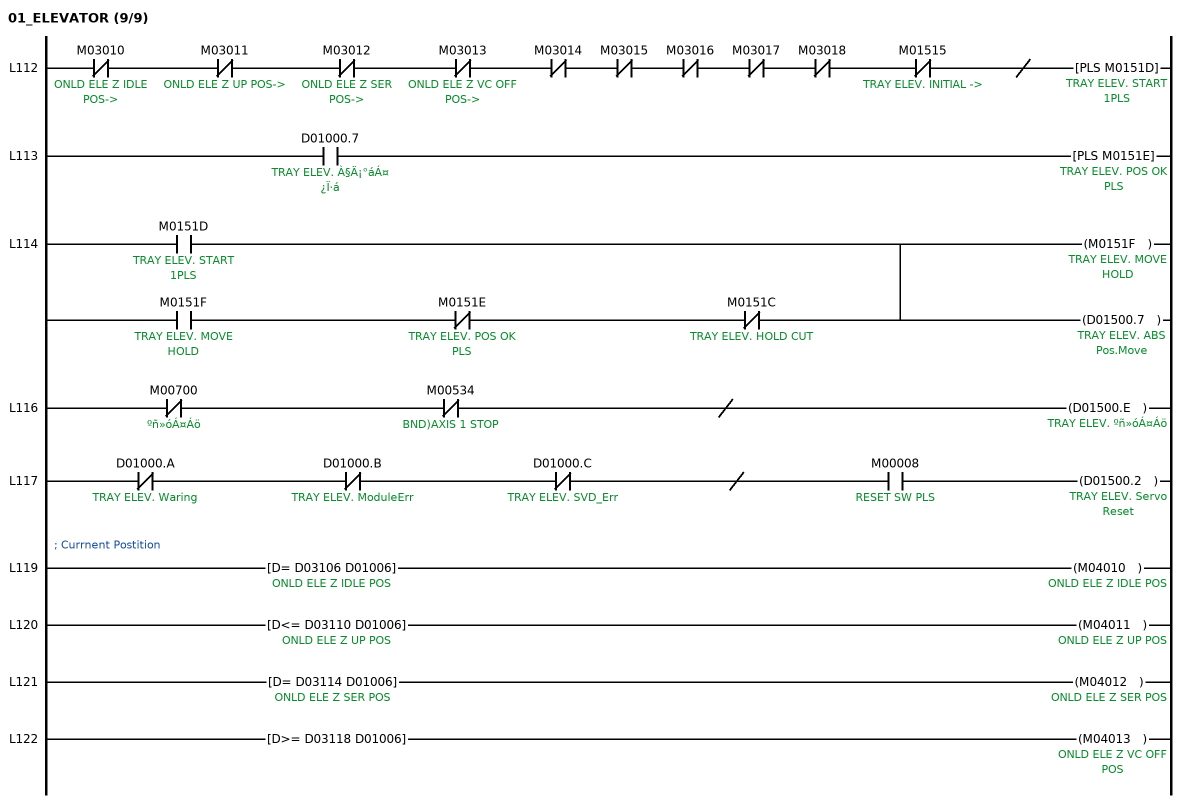
; L112
LOAD NOT  M03010	// ONLD ELE Z IDLE POS->
AND NOT   M03011	// ONLD ELE Z UP POS->
AND NOT   M03012	// ONLD ELE Z SER POS->
AND NOT   M03013	// ONLD ELE Z VC OFF POS->
AND NOT   M03014
AND NOT   M03015
AND NOT   M03016
AND NOT   M03017
AND NOT   M03018
AND NOT   M01515	// TRAY ELEV. INITIAL ->
NOT
OUTP      M0151D	// TRAY ELEV. START 1PLS
; L113
LOAD      D01000.7	// TRAY ELEV. À§Ä¡°áÁ¤ ¿Ï·á
OUTP      M0151E	// TRAY ELEV. POS OK PLS
; L114
LOAD      M0151D	// TRAY ELEV. START 1PLS
LOAD      M0151F	// TRAY ELEV. MOVE HOLD
AND NOT   M0151E	// TRAY ELEV. POS OK PLS
AND NOT   M0151C	// TRAY ELEV. HOLD CUT
OR LOAD
OUT       M0151F	// TRAY ELEV. MOVE HOLD
OUT       D01500.7	// TRAY ELEV. ABS Pos.Move
; L116
LOAD NOT  M00700	// ºñ»óÁ¤Áö
AND NOT   M00534	// BND)AXIS 1 STOP
NOT
OUT       D01500.E	// TRAY ELEV. ºñ»óÁ¤Áö
; L117
LOAD NOT  D01000.A	// TRAY ELEV. Waring
AND NOT   D01000.B	// TRAY ELEV. ModuleErr
AND NOT   D01000.C	// TRAY ELEV. SVD_Err
NOT
AND       M00008	// RESET SW PLS
OUT       D01500.2	// TRAY ELEV. Servo Reset
// Currnent Postition
; L119
LOADD=    D03106 D01006	// ONLD ELE Z IDLE POS
OUT       M04010	// ONLD ELE Z IDLE POS
; L120
LOADD<=   D03110 D01006	// ONLD ELE Z UP POS
OUT       M04011	// ONLD ELE Z UP POS
; L121
LOADD=    D03114 D01006	// ONLD ELE Z SER POS
OUT       M04012	// ONLD ELE Z SER POS
; L122
LOADD>=   D03118 D01006
OUT       M04013	// ONLD ELE Z VC OFF POS

PROGRAM 02_FEEDER_X1 (task: ½ºÄµ ÇÁ·Î±×·¥)

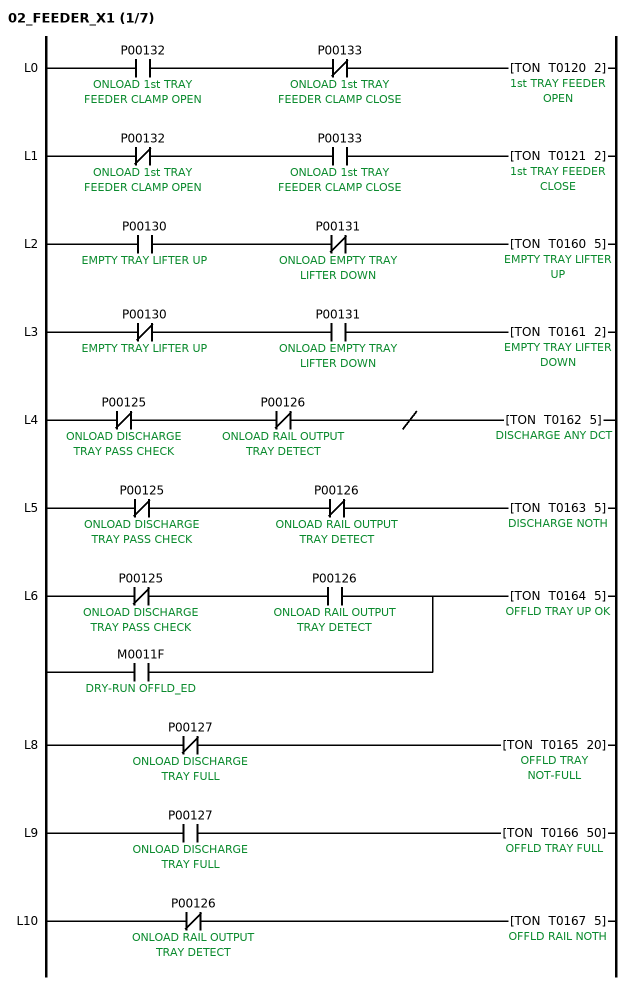
; L0
LOAD      P00132	// ONLOAD 1st TRAY FEEDER CLAMP OPEN
AND NOT   P00133	// ONLOAD 1st TRAY FEEDER CLAMP CLOSE
TON       T0120 2	// 1st TRAY FEEDER OPEN
; L1
LOAD NOT  P00132	// ONLOAD 1st TRAY FEEDER CLAMP OPEN
AND       P00133	// ONLOAD 1st TRAY FEEDER CLAMP CLOSE
TON       T0121 2	// 1st TRAY FEEDER CLOSE
; L2
LOAD      P00130	// EMPTY TRAY LIFTER UP
AND NOT   P00131	// ONLOAD EMPTY TRAY LIFTER DOWN
TON       T0160 5	// EMPTY TRAY LIFTER UP
; L3
LOAD NOT  P00130	// EMPTY TRAY LIFTER UP
AND       P00131	// ONLOAD EMPTY TRAY LIFTER DOWN
TON       T0161 2	// EMPTY TRAY LIFTER DOWN
; L4
LOAD NOT  P00125	// ONLOAD DISCHARGE TRAY PASS CHECK
AND NOT   P00126	// ONLOAD RAIL OUTPUT TRAY DETECT
NOT
TON       T0162 5	// DISCHARGE ANY DCT
; L5
LOAD NOT  P00125	// ONLOAD DISCHARGE TRAY PASS CHECK
AND NOT   P00126	// ONLOAD RAIL OUTPUT TRAY DETECT
TON       T0163 5	// DISCHARGE NOTH
; L6
LOAD NOT  P00125	// ONLOAD DISCHARGE TRAY PASS CHECK
AND       P00126	// ONLOAD RAIL OUTPUT TRAY DETECT
OR        M0011F	// DRY-RUN OFFLD_ED
TON       T0164 5	// OFFLD TRAY UP OK
; L8
LOAD NOT  P00127	// ONLOAD DISCHARGE TRAY FULL
TON       T0165 20	// OFFLD TRAY NOT-FULL
; L9
LOAD      P00127	// ONLOAD DISCHARGE TRAY FULL
TON       T0166 50	// OFFLD TRAY FULL
; L10
LOAD NOT  P00126	// ONLOAD RAIL OUTPUT TRAY DETECT
TON       T0167 5	// OFFLD RAIL NOTH

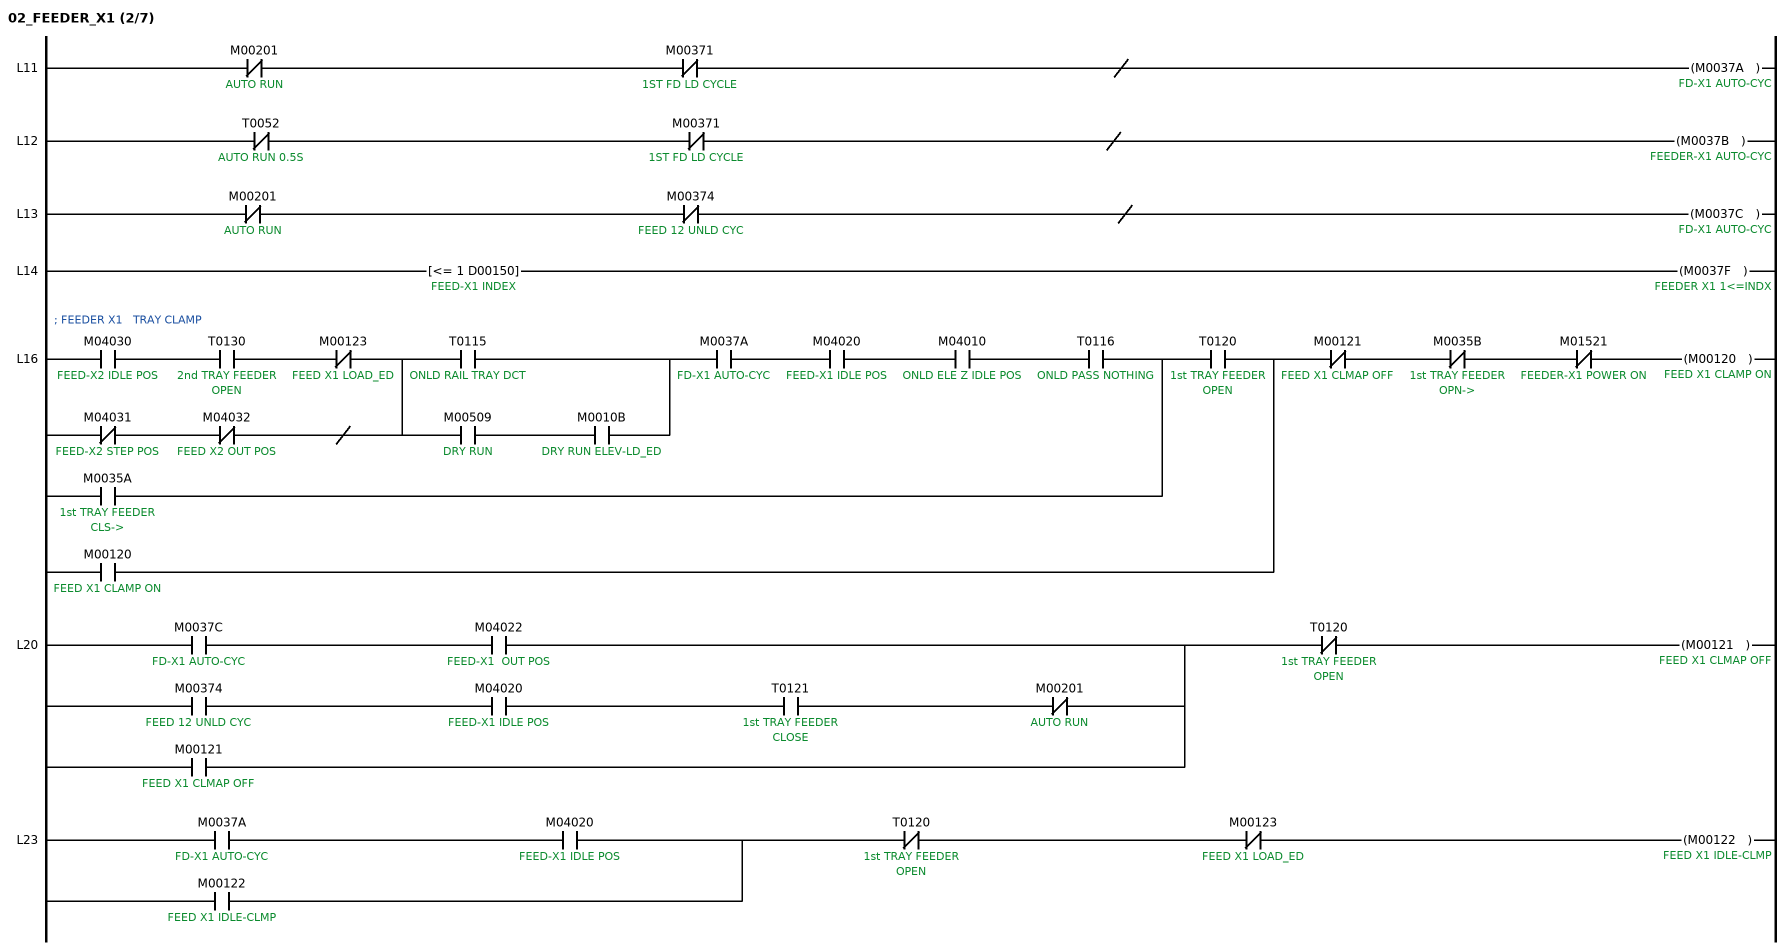
; L11
LOAD NOT  M00201	// AUTO RUN
AND NOT   M00371	// 1ST FD LD CYCLE
NOT
OUT       M0037A	// FD-X1 AUTO-CYC
; L12
LOAD NOT  T0052	// AUTO RUN 0.5S
AND NOT   M00371	// 1ST FD LD CYCLE
NOT
OUT       M0037B	// FEEDER-X1 AUTO-CYC
; L13
LOAD NOT  M00201	// AUTO RUN
AND NOT   M00374	// FEED 12 UNLD CYC
NOT
OUT       M0037C	// FD-X1 AUTO-CYC
; L14
LOAD<=    1 D00150	// FEED-X1 INDEX
OUT       M0037F	// FEEDER X1 1<=INDX
// FEEDER X1   TRAY CLAMP
; L16
LOAD      M04030	// FEED-X2 IDLE POS
AND       T0130	// 2nd TRAY FEEDER OPEN
AND NOT   M00123	// FEED X1 LOAD_ED
LOAD NOT  M04031	// FEED-X2 STEP POS
AND NOT   M04032	// FEED X2 OUT POS
NOT
OR LOAD
LOAD      T0115	// ONLD RAIL TRAY DCT
LOAD      M00509	// DRY RUN
AND       M0010B	// DRY RUN ELEV-LD_ED
OR LOAD
AND LOAD
AND       M0037A	// FD-X1 AUTO-CYC
AND       M04020	// FEED-X1 IDLE POS
AND       M04010	// ONLD ELE Z IDLE POS
AND       T0116	// ONLD PASS NOTHING
OR        M0035A	// 1st TRAY FEEDER CLS->
AND       T0120	// 1st TRAY FEEDER OPEN
OR        M00120	// FEED X1 CLAMP ON
AND NOT   M00121	// FEED X1 CLMAP OFF
AND NOT   M0035B	// 1st TRAY FEEDER OPN->
AND NOT   M01521	// FEEDER-X1 POWER ON
OUT       M00120	// FEED X1 CLAMP ON
; L20
LOAD      M0037C	// FD-X1 AUTO-CYC
AND       M04022	// FEED-X1  OUT POS
LOAD      M00374	// FEED 12 UNLD CYC
AND       M04020	// FEED-X1 IDLE POS
AND       T0121	// 1st TRAY FEEDER CLOSE
AND NOT   M00201	// AUTO RUN
OR LOAD
OR        M00121	// FEED X1 CLMAP OFF
AND NOT   T0120	// 1st TRAY FEEDER OPEN
OUT       M00121	// FEED X1 CLMAP OFF
; L23
LOAD      M0037A	// FD-X1 AUTO-CYC
AND       M04020	// FEED-X1 IDLE POS
OR        M00122	// FEED X1 IDLE-CLMP
AND NOT   T0120	// 1st TRAY FEEDER OPEN
AND NOT   M00123	// FEED X1 LOAD_ED
OUT       M00122	// FEED X1 IDLE-CLMP

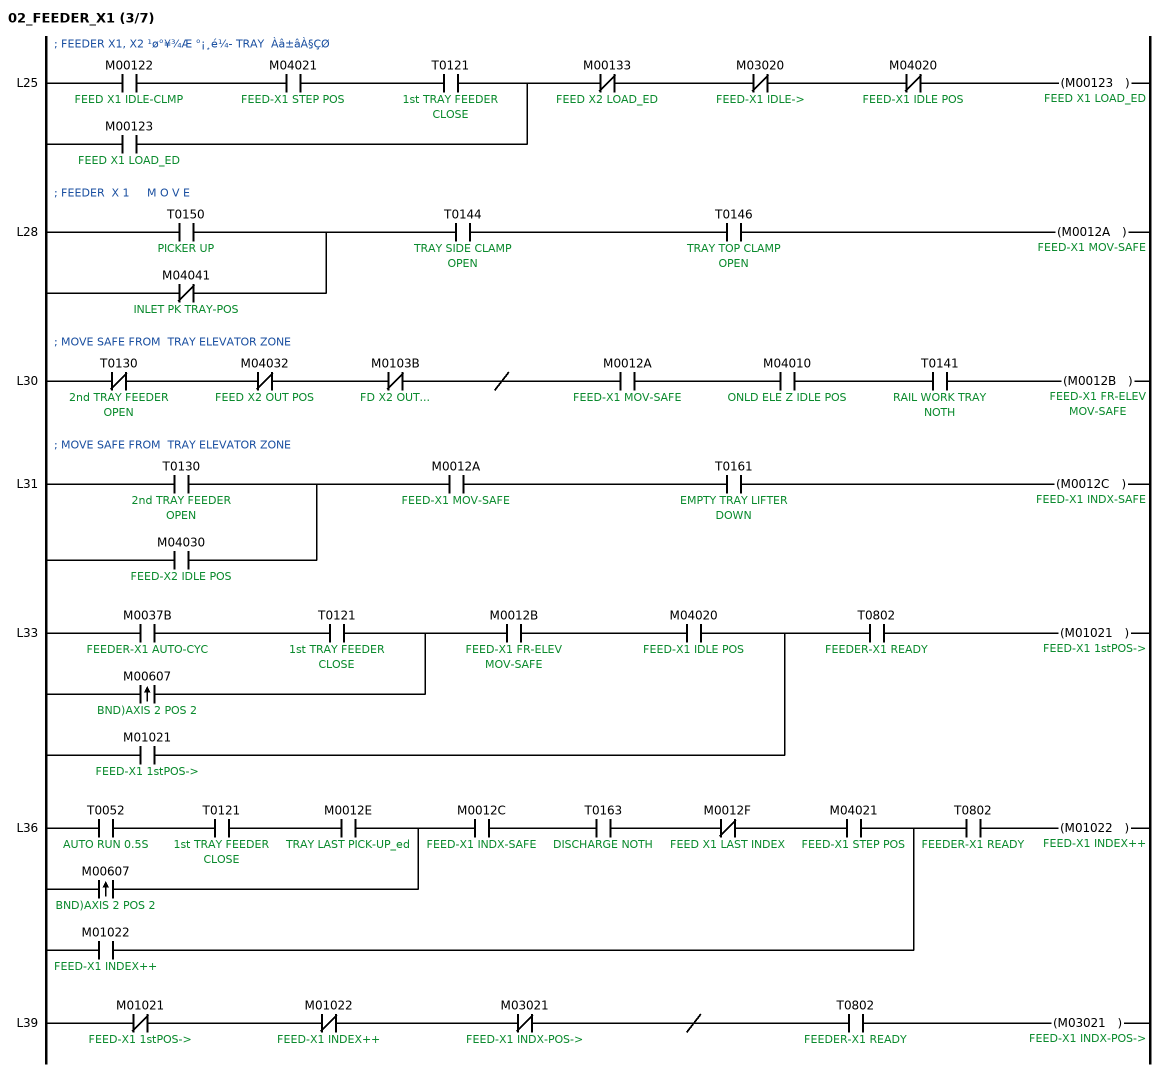
; L25
LOAD      M00122	// FEED X1 IDLE-CLMP
AND       M04021	// FEED-X1 STEP POS
AND       T0121	// 1st TRAY FEEDER CLOSE
OR        M00123	// FEED X1 LOAD_ED
AND NOT   M00133	// FEED X2 LOAD_ED
AND NOT   M03020	// FEED-X1 IDLE->
AND NOT   M04020	// FEED-X1 IDLE POS
OUT       M00123	// FEED X1 LOAD_ED
// output comment: FEEDER X1, X2 ¹ø°¥¾Æ °¡¸é¼­ TRAY  Àâ±âÀ§ÇØ
// FEEDER  X 1     M O V E
; L28
LOAD      T0150	// PICKER UP
OR NOT    M04041	// INLET PK TRAY-POS
AND       T0144	// TRAY SIDE CLAMP OPEN
AND       T0146	// TRAY TOP CLAMP OPEN
OUT       M0012A	// FEED-X1 MOV-SAFE
; L30
LOAD NOT  T0130	// 2nd TRAY FEEDER OPEN
AND NOT   M04032	// FEED X2 OUT POS
AND NOT   M0103B	// FD X2 OUT...
NOT
AND       M0012A	// FEED-X1 MOV-SAFE
AND       M04010	// ONLD ELE Z IDLE POS
AND       T0141	// RAIL WORK TRAY NOTH
OUT       M0012B	// FEED-X1 FR-ELEV MOV-SAFE
// output comment: MOVE SAFE FROM  TRAY ELEVATOR ZONE
; L31
LOAD      T0130	// 2nd TRAY FEEDER OPEN
OR        M04030	// FEED-X2 IDLE POS
AND       M0012A	// FEED-X1 MOV-SAFE
AND       T0161	// EMPTY TRAY LIFTER DOWN
OUT       M0012C	// FEED-X1 INDX-SAFE
// output comment: MOVE SAFE FROM  TRAY ELEVATOR ZONE
; L33
LOAD      M0037B	// FEEDER-X1 AUTO-CYC
AND       T0121	// 1st TRAY FEEDER CLOSE
ORP       M00607	// BND)AXIS 2 POS 2
AND       M0012B	// FEED-X1 FR-ELEV MOV-SAFE
AND       M04020	// FEED-X1 IDLE POS
OR        M01021	// FEED-X1 1stPOS->
AND       T0802	// FEEDER-X1 READY
OUT       M01021	// FEED-X1 1stPOS->
; L36
LOAD      T0052	// AUTO RUN 0.5S
AND       T0121	// 1st TRAY FEEDER CLOSE
AND       M0012E	// TRAY LAST PICK-UP_ed
ORP       M00607	// BND)AXIS 2 POS 2
AND       M0012C	// FEED-X1 INDX-SAFE
AND       T0163	// DISCHARGE NOTH
AND NOT   M0012F	// FEED X1 LAST INDEX
AND       M04021	// FEED-X1 STEP POS
OR        M01022	// FEED-X1 INDEX++
AND       T0802	// FEEDER-X1 READY
OUT       M01022	// FEED-X1 INDEX++
; L39
LOAD NOT  M01021	// FEED-X1 1stPOS->
AND NOT   M01022	// FEED-X1 INDEX++
AND NOT   M03021	// FEED-X1 INDX-POS->
NOT
AND       T0802	// FEEDER-X1 READY
OUT       M03021	// FEED-X1 INDX-POS->

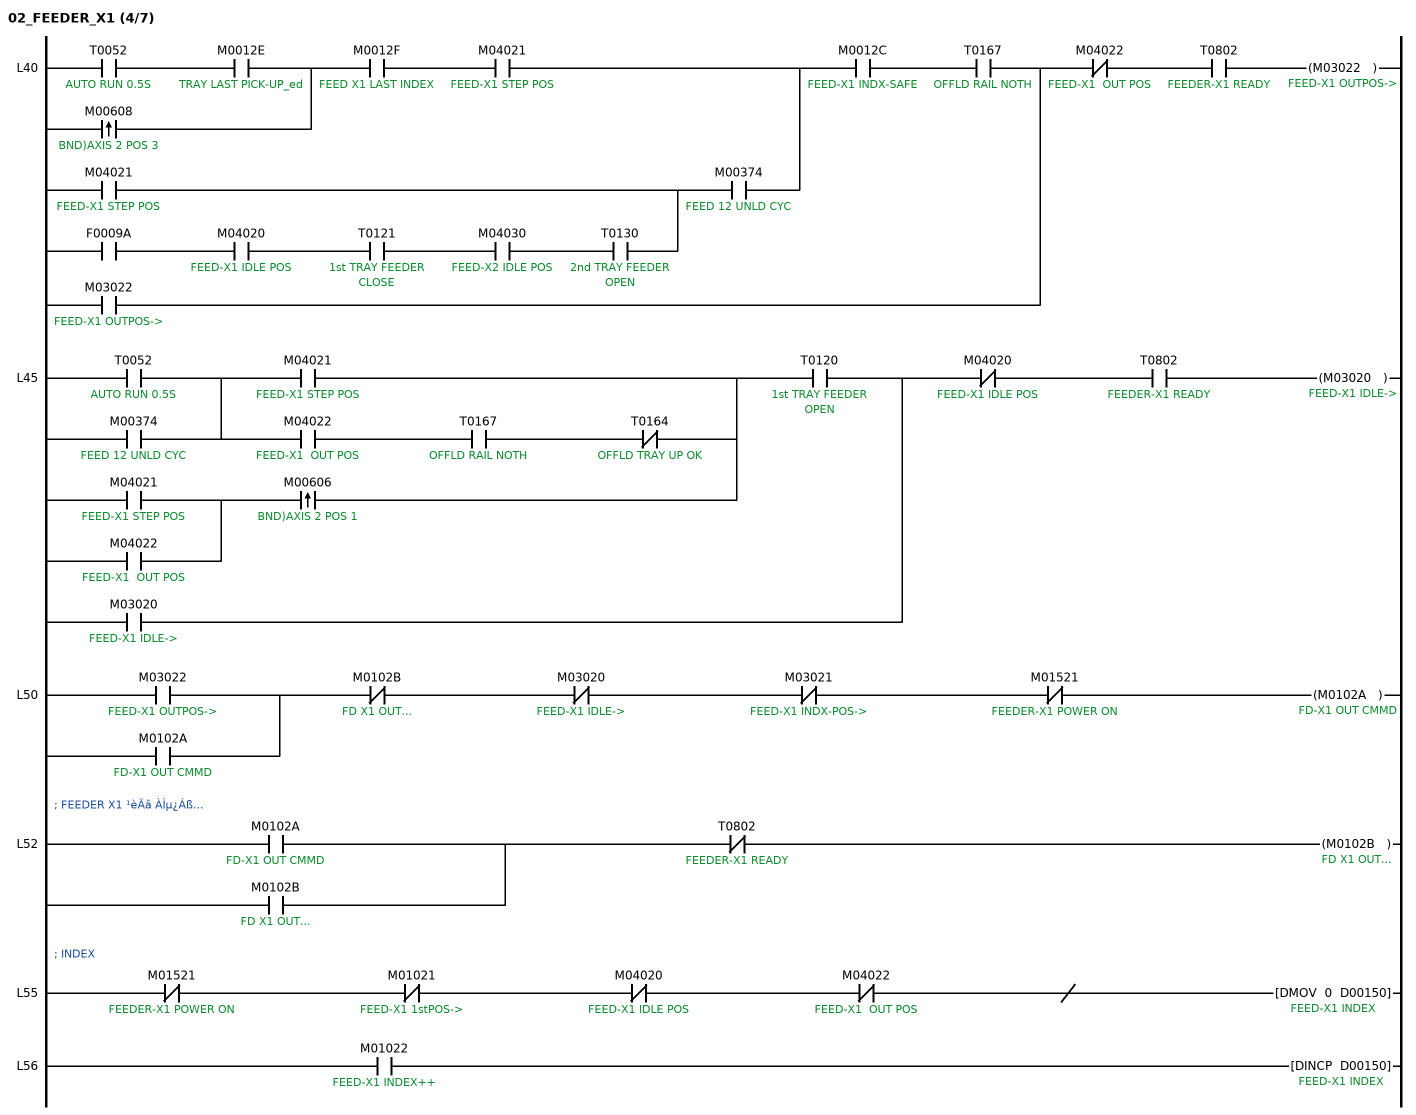
; L40
LOAD      T0052	// AUTO RUN 0.5S
AND       M0012E	// TRAY LAST PICK-UP_ed
ORP       M00608	// BND)AXIS 2 POS 3
AND       M0012F	// FEED X1 LAST INDEX
AND       M04021	// FEED-X1 STEP POS
LOAD      M04021	// FEED-X1 STEP POS
LOAD      F0009A
AND       M04020	// FEED-X1 IDLE POS
AND       T0121	// 1st TRAY FEEDER CLOSE
AND       M04030	// FEED-X2 IDLE POS
AND       T0130	// 2nd TRAY FEEDER OPEN
OR LOAD
AND       M00374	// FEED 12 UNLD CYC
OR LOAD
AND       M0012C	// FEED-X1 INDX-SAFE
AND       T0167	// OFFLD RAIL NOTH
OR        M03022	// FEED-X1 OUTPOS->
AND NOT   M04022	// FEED-X1  OUT POS
AND       T0802	// FEEDER-X1 READY
OUT       M03022	// FEED-X1 OUTPOS->
; L45
LOAD      T0052	// AUTO RUN 0.5S
OR        M00374	// FEED 12 UNLD CYC
LOAD      M04021	// FEED-X1 STEP POS
LOAD      M04022	// FEED-X1  OUT POS
AND       T0167	// OFFLD RAIL NOTH
AND NOT   T0164	// OFFLD TRAY UP OK
OR LOAD
AND LOAD
LOAD      M04021	// FEED-X1 STEP POS
OR        M04022	// FEED-X1  OUT POS
ANDP      M00606	// BND)AXIS 2 POS 1
OR LOAD
AND       T0120	// 1st TRAY FEEDER OPEN
OR        M03020	// FEED-X1 IDLE->
AND NOT   M04020	// FEED-X1 IDLE POS
AND       T0802	// FEEDER-X1 READY
OUT       M03020	// FEED-X1 IDLE->
; L50
LOAD      M03022	// FEED-X1 OUTPOS->
OR        M0102A	// FD-X1 OUT CMMD
AND NOT   M0102B	// FD X1 OUT...
AND NOT   M03020	// FEED-X1 IDLE->
AND NOT   M03021	// FEED-X1 INDX-POS->
AND NOT   M01521	// FEEDER-X1 POWER ON
OUT       M0102A	// FD-X1 OUT CMMD
; L52
LOAD      M0102A	// FD-X1 OUT CMMD
OR        M0102B	// FD X1 OUT...
AND NOT   T0802	// FEEDER-X1 READY
OUT       M0102B	// FD X1 OUT...
// output comment: FEEDER X1 ¹èÃâ ÀÌµ¿Áß...
// INDEX
; L55
LOAD NOT  M01521	// FEEDER-X1 POWER ON
AND NOT   M01021	// FEED-X1 1stPOS->
AND NOT   M04020	// FEED-X1 IDLE POS
AND NOT   M04022	// FEED-X1  OUT POS
NOT
DMOV      0 D00150	// FEED-X1 INDEX
; L56
LOAD      M01022	// FEED-X1 INDEX++
DINCP     D00150	// FEED-X1 INDEX

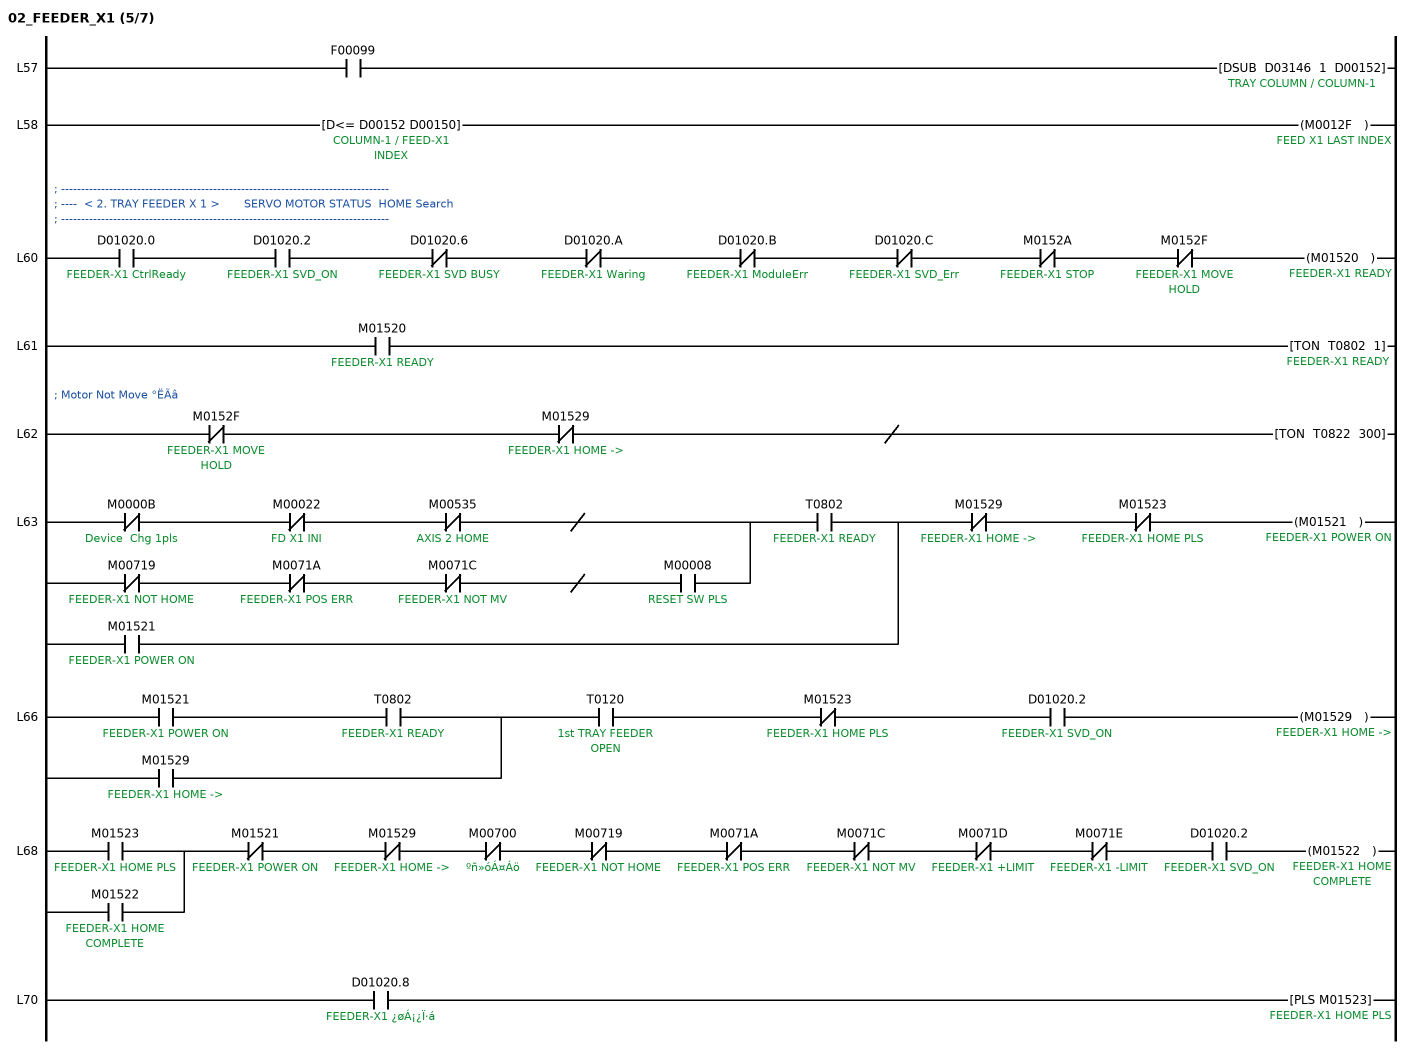
; L57
LOAD      F00099
DSUB      D03146 1 D00152	// TRAY COLUMN / COLUMN-1
; L58
LOADD<=   D00152 D00150	// COLUMN-1 / FEED-X1 INDEX
OUT       M0012F	// FEED X1 LAST INDEX
// ----------------------------------------------------------------------------------
// 
// ----  < 2. TRAY FEEDER X 1 >       SERVO MOTOR STATUS  HOME Search
// 
// ----------------------------------------------------------------------------------
; L60
LOAD      D01020.0	// FEEDER-X1 CtrlReady
AND       D01020.2	// FEEDER-X1 SVD_ON
AND NOT   D01020.6	// FEEDER-X1 SVD BUSY
AND NOT   D01020.A	// FEEDER-X1 Waring
AND NOT   D01020.B	// FEEDER-X1 ModuleErr
AND NOT   D01020.C	// FEEDER-X1 SVD_Err
AND NOT   M0152A	// FEEDER-X1 STOP
AND NOT   M0152F	// FEEDER-X1 MOVE HOLD
OUT       M01520	// FEEDER-X1 READY
; L61
LOAD      M01520	// FEEDER-X1 READY
TON       T0802 1	// FEEDER-X1 READY
; L62
LOAD NOT  M0152F	// FEEDER-X1 MOVE HOLD
AND NOT   M01529	// FEEDER-X1 HOME ->
NOT
TON       T0822 300
// output comment: Motor Not Move °ËÃâ
; L63
LOAD NOT  M0000B	// Device  Chg 1pls
AND NOT   M00022	// FD X1 INI
AND NOT   M00535	// AXIS 2 HOME
NOT
LOAD NOT  M00719	// FEEDER-X1 NOT HOME
AND NOT   M0071A	// FEEDER-X1 POS ERR
AND NOT   M0071C	// FEEDER-X1 NOT MV
NOT
AND       M00008	// RESET SW PLS
OR LOAD
AND       T0802	// FEEDER-X1 READY
OR        M01521	// FEEDER-X1 POWER ON
AND NOT   M01529	// FEEDER-X1 HOME ->
AND NOT   M01523	// FEEDER-X1 HOME PLS
OUT       M01521	// FEEDER-X1 POWER ON
; L66
LOAD      M01521	// FEEDER-X1 POWER ON
AND       T0802	// FEEDER-X1 READY
OR        M01529	// FEEDER-X1 HOME ->
AND       T0120	// 1st TRAY FEEDER OPEN
AND NOT   M01523	// FEEDER-X1 HOME PLS
AND       D01020.2	// FEEDER-X1 SVD_ON
OUT       M01529	// FEEDER-X1 HOME ->
; L68
LOAD      M01523	// FEEDER-X1 HOME PLS
OR        M01522	// FEEDER-X1 HOME COMPLETE
AND NOT   M01521	// FEEDER-X1 POWER ON
AND NOT   M01529	// FEEDER-X1 HOME ->
AND NOT   M00700	// ºñ»óÁ¤Áö
AND NOT   M00719	// FEEDER-X1 NOT HOME
AND NOT   M0071A	// FEEDER-X1 POS ERR
AND NOT   M0071C	// FEEDER-X1 NOT MV
AND NOT   M0071D	// FEEDER-X1 +LIMIT
AND NOT   M0071E	// FEEDER-X1 -LIMIT
AND       D01020.2	// FEEDER-X1 SVD_ON
OUT       M01522	// FEEDER-X1 HOME COMPLETE
; L70
LOAD      D01020.8	// FEEDER-X1 ¿øÁ¡¿Ï·á
OUTP      M01523	// FEEDER-X1 HOME PLS

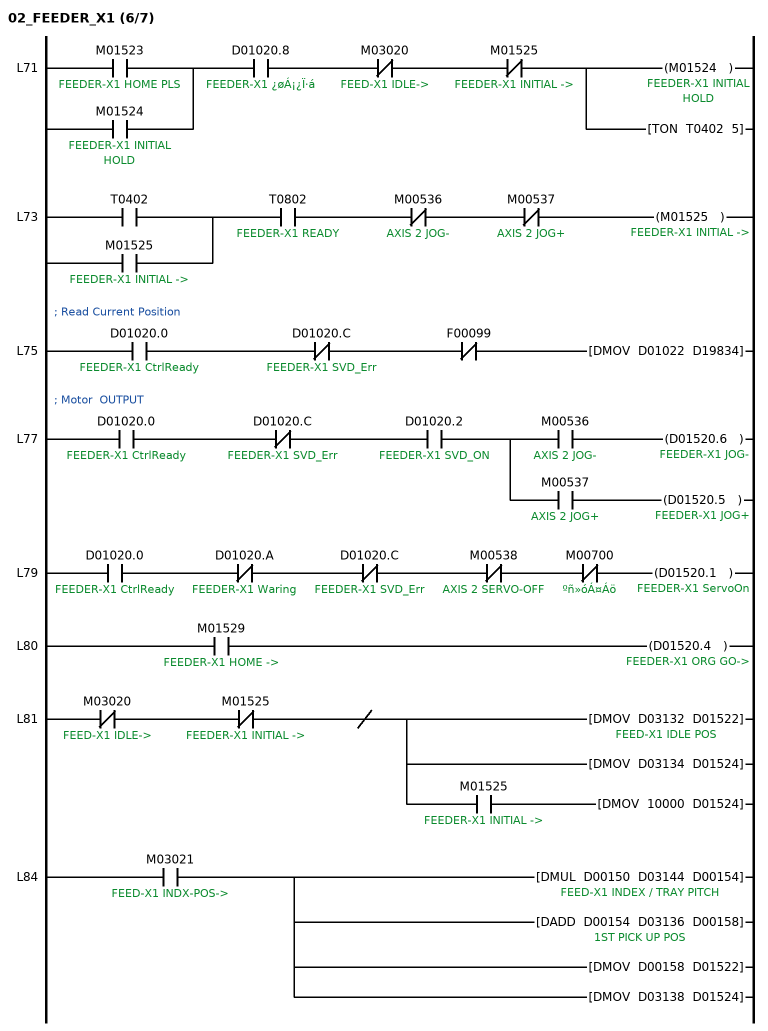
; L71
LOAD      M01523	// FEEDER-X1 HOME PLS
OR        M01524	// FEEDER-X1 INITIAL HOLD
AND       D01020.8	// FEEDER-X1 ¿øÁ¡¿Ï·á
AND NOT   M03020	// FEED-X1 IDLE->
AND NOT   M01525	// FEEDER-X1 INITIAL ->
OUT       M01524	// FEEDER-X1 INITIAL HOLD
TON       T0402 5
; L73
LOAD      T0402
OR        M01525	// FEEDER-X1 INITIAL ->
AND       T0802	// FEEDER-X1 READY
AND NOT   M00536	// AXIS 2 JOG-
AND NOT   M00537	// AXIS 2 JOG+
OUT       M01525	// FEEDER-X1 INITIAL ->
; L75
LOAD      D01020.0	// FEEDER-X1 CtrlReady
AND NOT   D01020.C	// FEEDER-X1 SVD_Err
AND NOT   F00099
DMOV      D01022 D19834
// output comment: Read Current Position
//  Motor  OUTPUT
; L77
LOAD      D01020.0	// FEEDER-X1 CtrlReady
AND NOT   D01020.C	// FEEDER-X1 SVD_Err
AND       D01020.2	// FEEDER-X1 SVD_ON
MPUSH
AND       M00536	// AXIS 2 JOG-
OUT       D01520.6	// FEEDER-X1 JOG-
MPOP
AND       M00537	// AXIS 2 JOG+
OUT       D01520.5	// FEEDER-X1 JOG+
; L79
LOAD      D01020.0	// FEEDER-X1 CtrlReady
AND NOT   D01020.A	// FEEDER-X1 Waring
AND NOT   D01020.C	// FEEDER-X1 SVD_Err
AND NOT   M00538	// AXIS 2 SERVO-OFF
AND NOT   M00700	// ºñ»óÁ¤Áö
OUT       D01520.1	// FEEDER-X1 ServoOn
; L80
LOAD      M01529	// FEEDER-X1 HOME ->
OUT       D01520.4	// FEEDER-X1 ORG GO->
; L81
LOAD NOT  M03020	// FEED-X1 IDLE->
AND NOT   M01525	// FEEDER-X1 INITIAL ->
NOT
DMOV      D03132 D01522	// FEED-X1 IDLE POS
DMOV      D03134 D01524
AND       M01525	// FEEDER-X1 INITIAL ->
DMOV      10000 D01524
; L84
LOAD      M03021	// FEED-X1 INDX-POS->
DMUL      D00150 D03144 D00154	// FEED-X1 INDEX / TRAY PITCH
DADD      D00154 D03136 D00158	// 1ST PICK UP POS
DMOV      D00158 D01522
DMOV      D03138 D01524

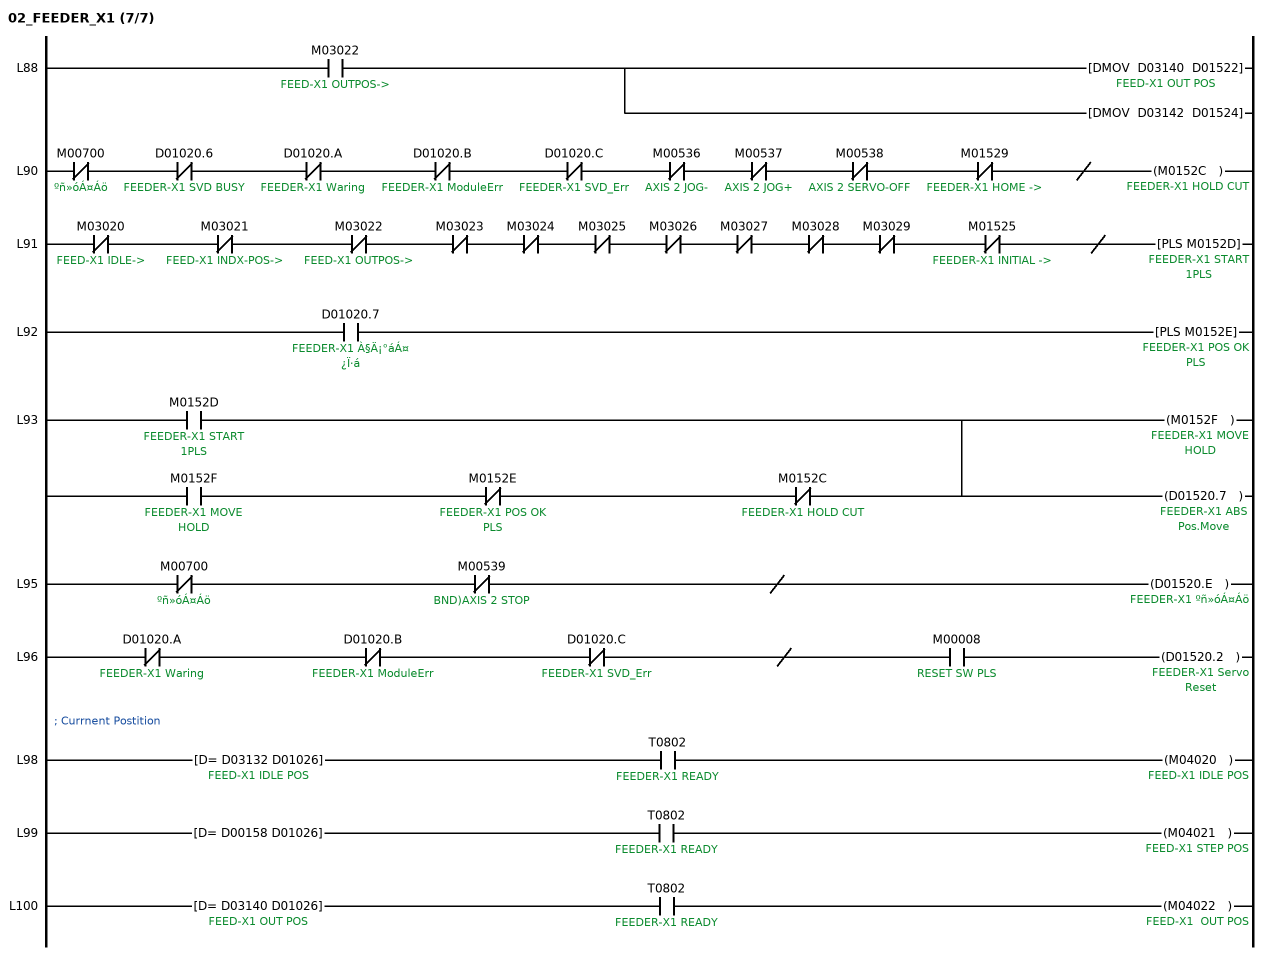
; L88
LOAD      M03022	// FEED-X1 OUTPOS->
DMOV      D03140 D01522	// FEED-X1 OUT POS
DMOV      D03142 D01524
; L90
LOAD NOT  M00700	// ºñ»óÁ¤Áö
AND NOT   D01020.6	// FEEDER-X1 SVD BUSY
AND NOT   D01020.A	// FEEDER-X1 Waring
AND NOT   D01020.B	// FEEDER-X1 ModuleErr
AND NOT   D01020.C	// FEEDER-X1 SVD_Err
AND NOT   M00536	// AXIS 2 JOG-
AND NOT   M00537	// AXIS 2 JOG+
AND NOT   M00538	// AXIS 2 SERVO-OFF
AND NOT   M01529	// FEEDER-X1 HOME ->
NOT
OUT       M0152C	// FEEDER-X1 HOLD CUT
; L91
LOAD NOT  M03020	// FEED-X1 IDLE->
AND NOT   M03021	// FEED-X1 INDX-POS->
AND NOT   M03022	// FEED-X1 OUTPOS->
AND NOT   M03023
AND NOT   M03024
AND NOT   M03025
AND NOT   M03026
AND NOT   M03027
AND NOT   M03028
AND NOT   M03029
AND NOT   M01525	// FEEDER-X1 INITIAL ->
NOT
OUTP      M0152D	// FEEDER-X1 START 1PLS
; L92
LOAD      D01020.7	// FEEDER-X1 À§Ä¡°áÁ¤ ¿Ï·á
OUTP      M0152E	// FEEDER-X1 POS OK PLS
; L93
LOAD      M0152D	// FEEDER-X1 START 1PLS
LOAD      M0152F	// FEEDER-X1 MOVE HOLD
AND NOT   M0152E	// FEEDER-X1 POS OK PLS
AND NOT   M0152C	// FEEDER-X1 HOLD CUT
OR LOAD
OUT       M0152F	// FEEDER-X1 MOVE HOLD
OUT       D01520.7	// FEEDER-X1 ABS Pos.Move
; L95
LOAD NOT  M00700	// ºñ»óÁ¤Áö
AND NOT   M00539	// BND)AXIS 2 STOP
NOT
OUT       D01520.E	// FEEDER-X1 ºñ»óÁ¤Áö
; L96
LOAD NOT  D01020.A	// FEEDER-X1 Waring
AND NOT   D01020.B	// FEEDER-X1 ModuleErr
AND NOT   D01020.C	// FEEDER-X1 SVD_Err
NOT
AND       M00008	// RESET SW PLS
OUT       D01520.2	// FEEDER-X1 Servo Reset
// Currnent Postition
; L98
LOADD=    D03132 D01026	// FEED-X1 IDLE POS
AND       T0802	// FEEDER-X1 READY
OUT       M04020	// FEED-X1 IDLE POS
; L99
LOADD=    D00158 D01026
AND       T0802	// FEEDER-X1 READY
OUT       M04021	// FEED-X1 STEP POS
; L100
LOADD=    D03140 D01026	// FEED-X1 OUT POS
AND       T0802	// FEEDER-X1 READY
OUT       M04022	// FEED-X1  OUT POS

PROGRAM 03_FEEDER_X2 (task: ½ºÄµ ÇÁ·Î±×·¥)

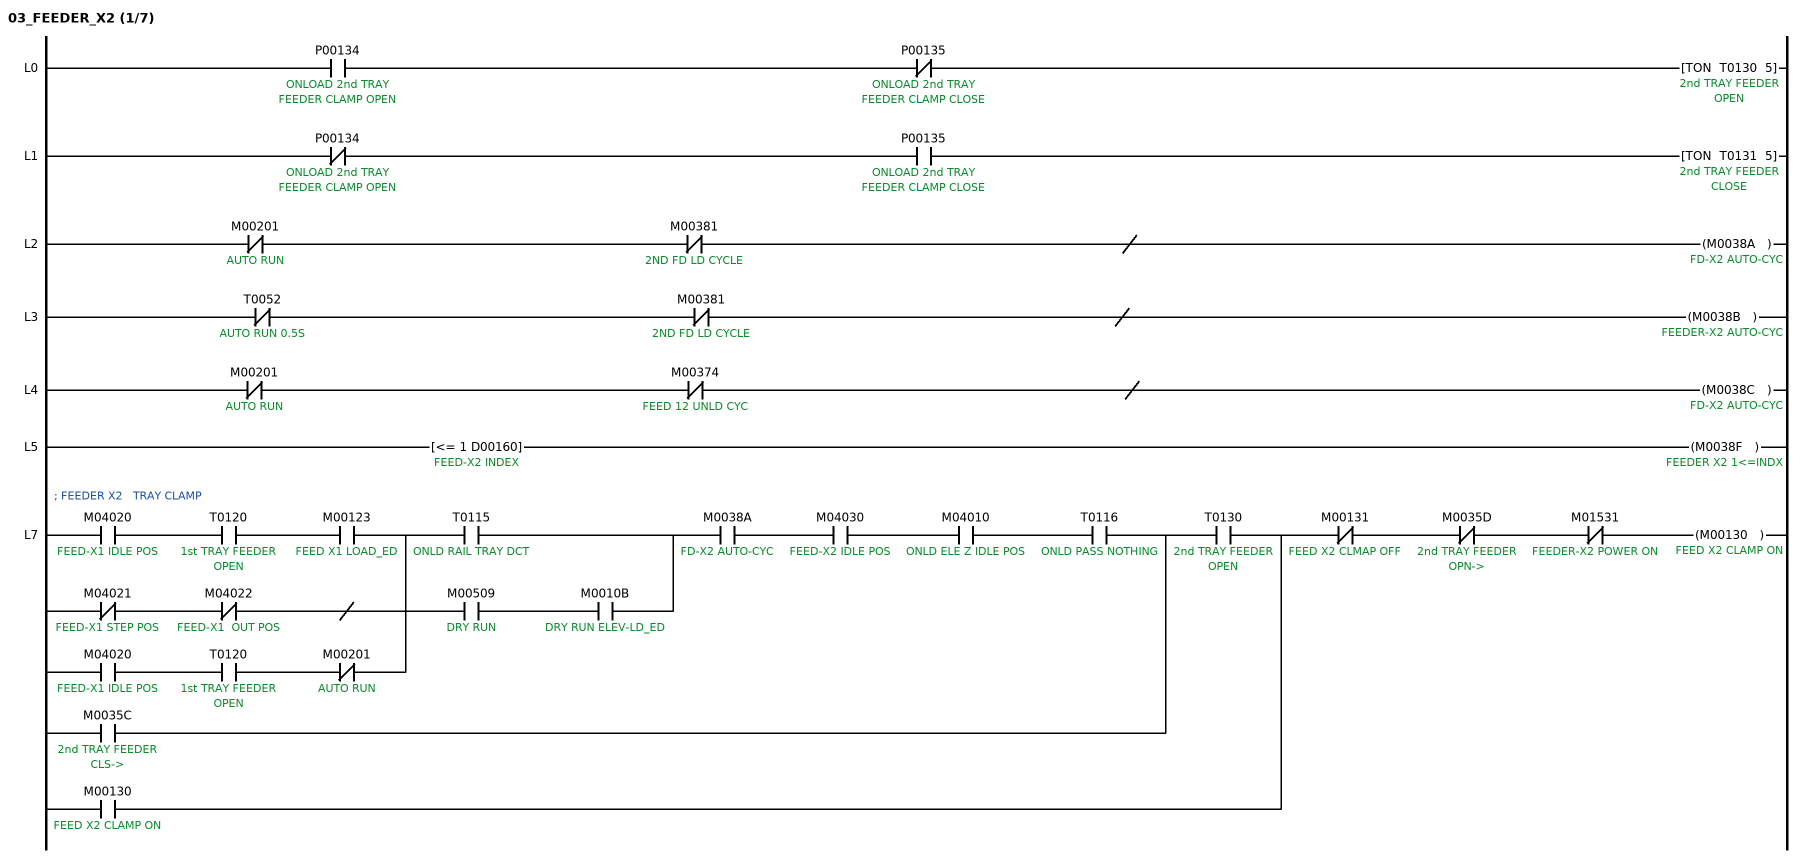
; L0
LOAD      P00134	// ONLOAD 2nd TRAY FEEDER CLAMP OPEN
AND NOT   P00135	// ONLOAD 2nd TRAY FEEDER CLAMP CLOSE
TON       T0130 5	// 2nd TRAY FEEDER OPEN
; L1
LOAD NOT  P00134	// ONLOAD 2nd TRAY FEEDER CLAMP OPEN
AND       P00135	// ONLOAD 2nd TRAY FEEDER CLAMP CLOSE
TON       T0131 5	// 2nd TRAY FEEDER CLOSE
; L2
LOAD NOT  M00201	// AUTO RUN
AND NOT   M00381	// 2ND FD LD CYCLE
NOT
OUT       M0038A	// FD-X2 AUTO-CYC
; L3
LOAD NOT  T0052	// AUTO RUN 0.5S
AND NOT   M00381	// 2ND FD LD CYCLE
NOT
OUT       M0038B	// FEEDER-X2 AUTO-CYC
; L4
LOAD NOT  M00201	// AUTO RUN
AND NOT   M00374	// FEED 12 UNLD CYC
NOT
OUT       M0038C	// FD-X2 AUTO-CYC
; L5
LOAD<=    1 D00160	// FEED-X2 INDEX
OUT       M0038F	// FEEDER X2 1<=INDX
// FEEDER X2   TRAY CLAMP
; L7
LOAD      M04020	// FEED-X1 IDLE POS
AND       T0120	// 1st TRAY FEEDER OPEN
AND       M00123	// FEED X1 LOAD_ED
LOAD NOT  M04021	// FEED-X1 STEP POS
AND NOT   M04022	// FEED-X1  OUT POS
NOT
OR LOAD
LOAD      M04020	// FEED-X1 IDLE POS
AND       T0120	// 1st TRAY FEEDER OPEN
AND NOT   M00201	// AUTO RUN
OR LOAD
LOAD      T0115	// ONLD RAIL TRAY DCT
LOAD      M00509	// DRY RUN
AND       M0010B	// DRY RUN ELEV-LD_ED
OR LOAD
AND LOAD
AND       M0038A	// FD-X2 AUTO-CYC
AND       M04030	// FEED-X2 IDLE POS
AND       M04010	// ONLD ELE Z IDLE POS
AND       T0116	// ONLD PASS NOTHING
OR        M0035C	// 2nd TRAY FEEDER CLS->
AND       T0130	// 2nd TRAY FEEDER OPEN
OR        M00130	// FEED X2 CLAMP ON
AND NOT   M00131	// FEED X2 CLMAP OFF
AND NOT   M0035D	// 2nd TRAY FEEDER OPN->
AND NOT   M01531	// FEEDER-X2 POWER ON
OUT       M00130	// FEED X2 CLAMP ON

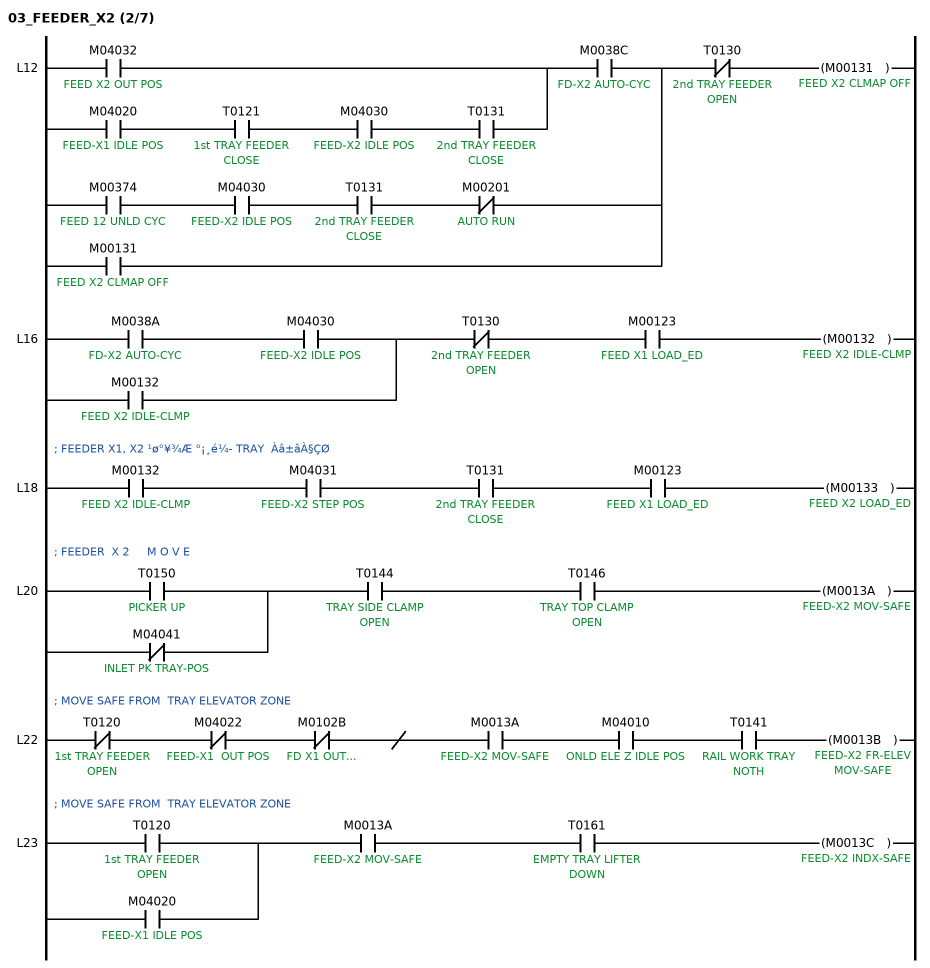
; L12
LOAD      M04032	// FEED X2 OUT POS
LOAD      M04020	// FEED-X1 IDLE POS
AND       T0121	// 1st TRAY FEEDER CLOSE
AND       M04030	// FEED-X2 IDLE POS
AND       T0131	// 2nd TRAY FEEDER CLOSE
OR LOAD
AND       M0038C	// FD-X2 AUTO-CYC
LOAD      M00374	// FEED 12 UNLD CYC
AND       M04030	// FEED-X2 IDLE POS
AND       T0131	// 2nd TRAY FEEDER CLOSE
AND NOT   M00201	// AUTO RUN
OR LOAD
OR        M00131	// FEED X2 CLMAP OFF
AND NOT   T0130	// 2nd TRAY FEEDER OPEN
OUT       M00131	// FEED X2 CLMAP OFF
; L16
LOAD      M0038A	// FD-X2 AUTO-CYC
AND       M04030	// FEED-X2 IDLE POS
OR        M00132	// FEED X2 IDLE-CLMP
AND NOT   T0130	// 2nd TRAY FEEDER OPEN
AND       M00123	// FEED X1 LOAD_ED
OUT       M00132	// FEED X2 IDLE-CLMP
; L18
LOAD      M00132	// FEED X2 IDLE-CLMP
AND       M04031	// FEED-X2 STEP POS
AND       T0131	// 2nd TRAY FEEDER CLOSE
AND       M00123	// FEED X1 LOAD_ED
OUT       M00133	// FEED X2 LOAD_ED
// output comment: FEEDER X1, X2 ¹ø°¥¾Æ °¡¸é¼­ TRAY  Àâ±âÀ§ÇØ
// FEEDER  X 2     M O V E
; L20
LOAD      T0150	// PICKER UP
OR NOT    M04041	// INLET PK TRAY-POS
AND       T0144	// TRAY SIDE CLAMP OPEN
AND       T0146	// TRAY TOP CLAMP OPEN
OUT       M0013A	// FEED-X2 MOV-SAFE
; L22
LOAD NOT  T0120	// 1st TRAY FEEDER OPEN
AND NOT   M04022	// FEED-X1  OUT POS
AND NOT   M0102B	// FD X1 OUT...
NOT
AND       M0013A	// FEED-X2 MOV-SAFE
AND       M04010	// ONLD ELE Z IDLE POS
AND       T0141	// RAIL WORK TRAY NOTH
OUT       M0013B	// FEED-X2 FR-ELEV MOV-SAFE
// output comment: MOVE SAFE FROM  TRAY ELEVATOR ZONE
; L23
LOAD      T0120	// 1st TRAY FEEDER OPEN
OR        M04020	// FEED-X1 IDLE POS
AND       M0013A	// FEED-X2 MOV-SAFE
AND       T0161	// EMPTY TRAY LIFTER DOWN
OUT       M0013C	// FEED-X2 INDX-SAFE
// output comment: MOVE SAFE FROM  TRAY ELEVATOR ZONE

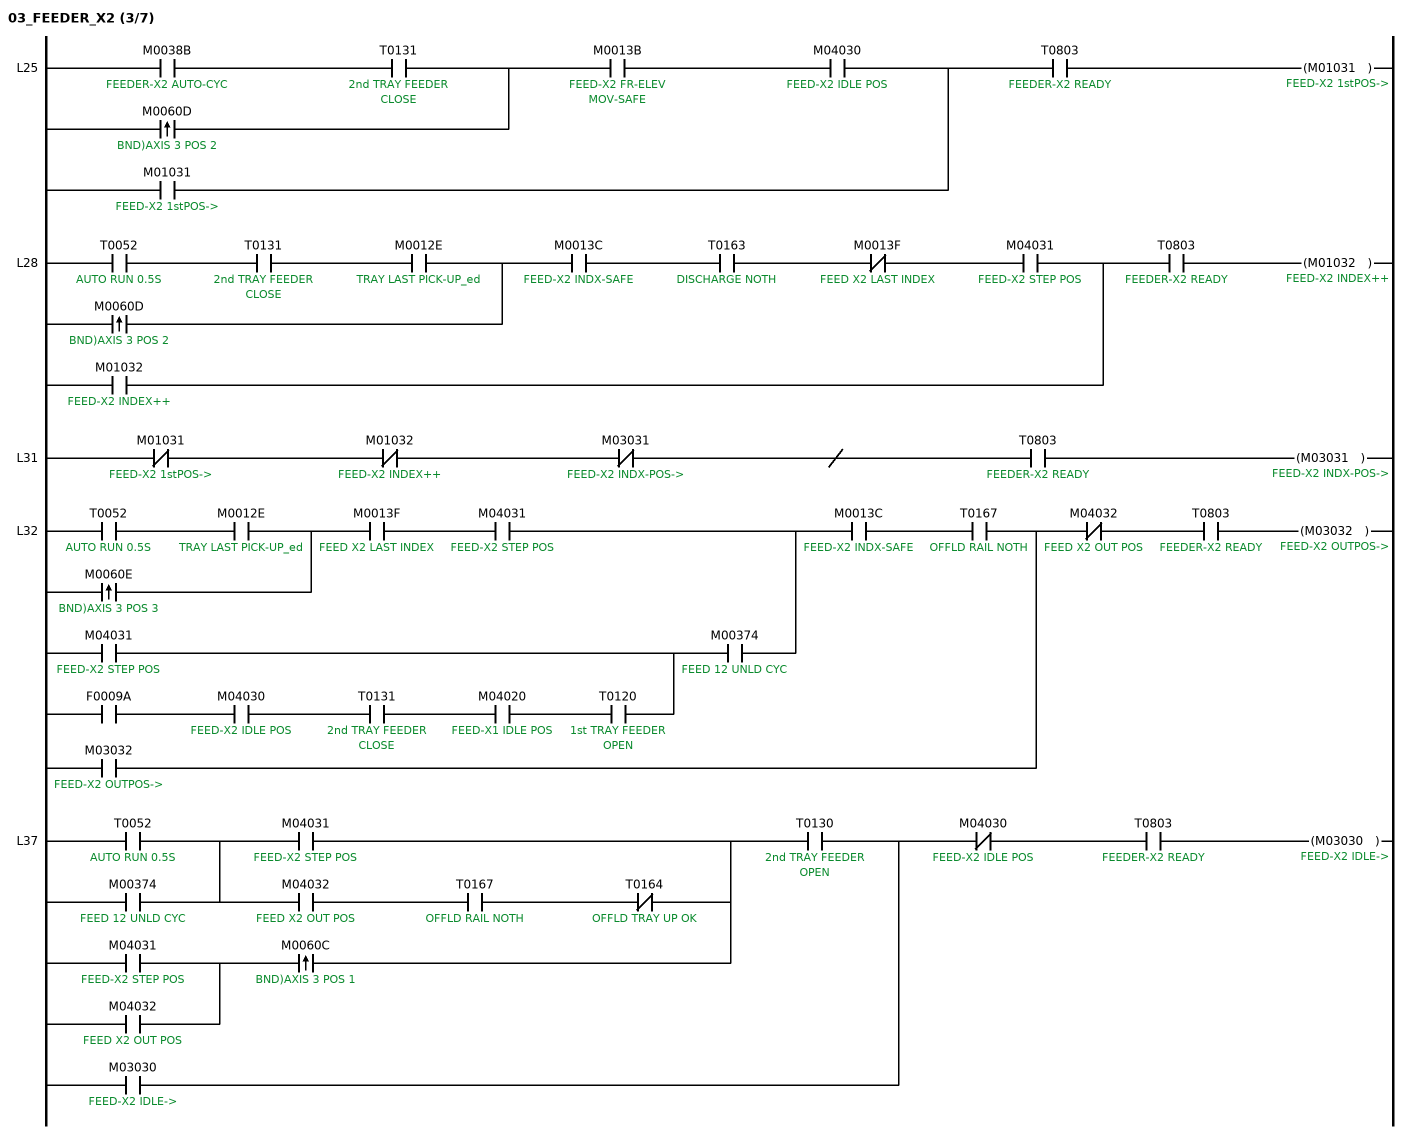
; L25
LOAD      M0038B	// FEEDER-X2 AUTO-CYC
AND       T0131	// 2nd TRAY FEEDER CLOSE
ORP       M0060D	// BND)AXIS 3 POS 2
AND       M0013B	// FEED-X2 FR-ELEV MOV-SAFE
AND       M04030	// FEED-X2 IDLE POS
OR        M01031	// FEED-X2 1stPOS->
AND       T0803	// FEEDER-X2 READY
OUT       M01031	// FEED-X2 1stPOS->
; L28
LOAD      T0052	// AUTO RUN 0.5S
AND       T0131	// 2nd TRAY FEEDER CLOSE
AND       M0012E	// TRAY LAST PICK-UP_ed
ORP       M0060D	// BND)AXIS 3 POS 2
AND       M0013C	// FEED-X2 INDX-SAFE
AND       T0163	// DISCHARGE NOTH
AND NOT   M0013F	// FEED X2 LAST INDEX
AND       M04031	// FEED-X2 STEP POS
OR        M01032	// FEED-X2 INDEX++
AND       T0803	// FEEDER-X2 READY
OUT       M01032	// FEED-X2 INDEX++
; L31
LOAD NOT  M01031	// FEED-X2 1stPOS->
AND NOT   M01032	// FEED-X2 INDEX++
AND NOT   M03031	// FEED-X2 INDX-POS->
NOT
AND       T0803	// FEEDER-X2 READY
OUT       M03031	// FEED-X2 INDX-POS->
; L32
LOAD      T0052	// AUTO RUN 0.5S
AND       M0012E	// TRAY LAST PICK-UP_ed
ORP       M0060E	// BND)AXIS 3 POS 3
AND       M0013F	// FEED X2 LAST INDEX
AND       M04031	// FEED-X2 STEP POS
LOAD      M04031	// FEED-X2 STEP POS
LOAD      F0009A
AND       M04030	// FEED-X2 IDLE POS
AND       T0131	// 2nd TRAY FEEDER CLOSE
AND       M04020	// FEED-X1 IDLE POS
AND       T0120	// 1st TRAY FEEDER OPEN
OR LOAD
AND       M00374	// FEED 12 UNLD CYC
OR LOAD
AND       M0013C	// FEED-X2 INDX-SAFE
AND       T0167	// OFFLD RAIL NOTH
OR        M03032	// FEED-X2 OUTPOS->
AND NOT   M04032	// FEED X2 OUT POS
AND       T0803	// FEEDER-X2 READY
OUT       M03032	// FEED-X2 OUTPOS->
; L37
LOAD      T0052	// AUTO RUN 0.5S
OR        M00374	// FEED 12 UNLD CYC
LOAD      M04031	// FEED-X2 STEP POS
LOAD      M04032	// FEED X2 OUT POS
AND       T0167	// OFFLD RAIL NOTH
AND NOT   T0164	// OFFLD TRAY UP OK
OR LOAD
AND LOAD
LOAD      M04031	// FEED-X2 STEP POS
OR        M04032	// FEED X2 OUT POS
ANDP      M0060C	// BND)AXIS 3 POS 1
OR LOAD
AND       T0130	// 2nd TRAY FEEDER OPEN
OR        M03030	// FEED-X2 IDLE->
AND NOT   M04030	// FEED-X2 IDLE POS
AND       T0803	// FEEDER-X2 READY
OUT       M03030	// FEED-X2 IDLE->

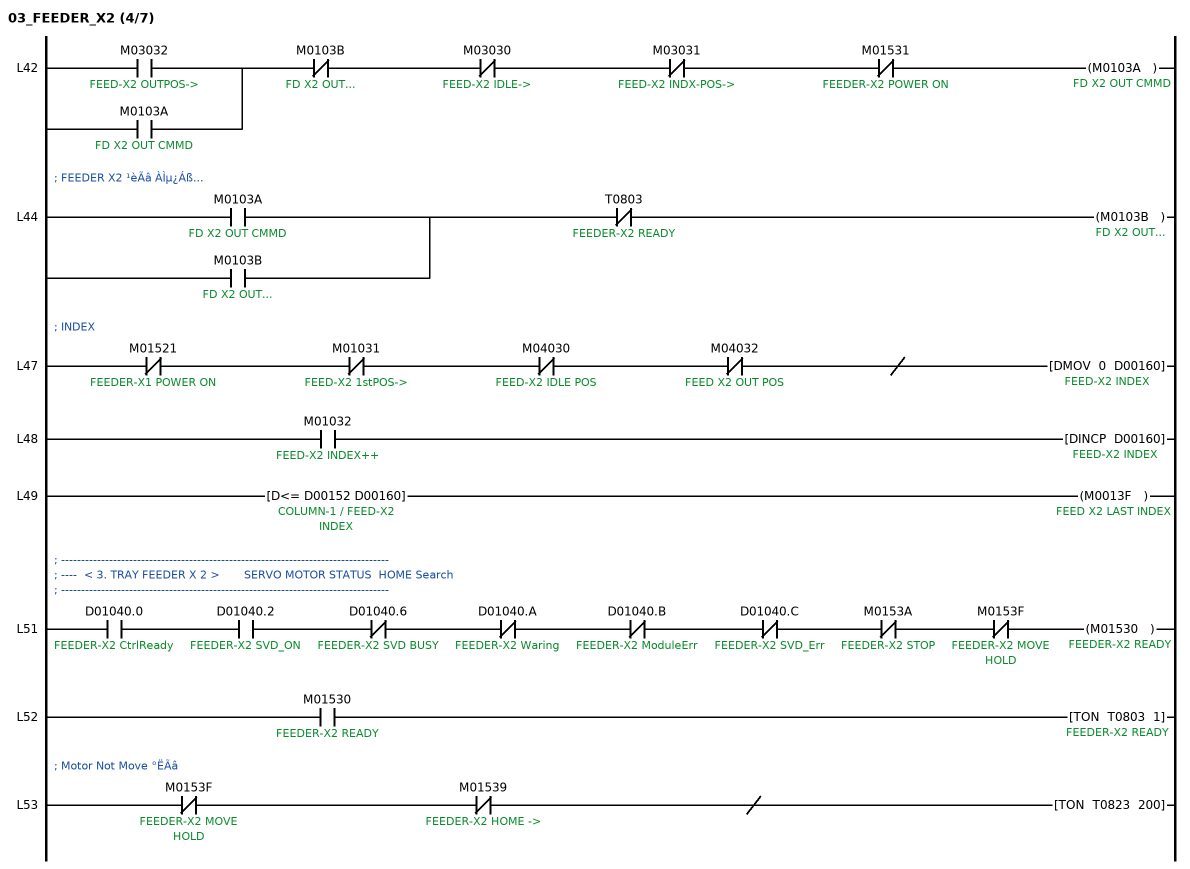
; L42
LOAD      M03032	// FEED-X2 OUTPOS->
OR        M0103A	// FD X2 OUT CMMD
AND NOT   M0103B	// FD X2 OUT...
AND NOT   M03030	// FEED-X2 IDLE->
AND NOT   M03031	// FEED-X2 INDX-POS->
AND NOT   M01531	// FEEDER-X2 POWER ON
OUT       M0103A	// FD X2 OUT CMMD
; L44
LOAD      M0103A	// FD X2 OUT CMMD
OR        M0103B	// FD X2 OUT...
AND NOT   T0803	// FEEDER-X2 READY
OUT       M0103B	// FD X2 OUT...
// output comment: FEEDER X2 ¹èÃâ ÀÌµ¿Áß...
// INDEX
; L47
LOAD NOT  M01521	// FEEDER-X1 POWER ON
AND NOT   M01031	// FEED-X2 1stPOS->
AND NOT   M04030	// FEED-X2 IDLE POS
AND NOT   M04032	// FEED X2 OUT POS
NOT
DMOV      0 D00160	// FEED-X2 INDEX
; L48
LOAD      M01032	// FEED-X2 INDEX++
DINCP     D00160	// FEED-X2 INDEX
; L49
LOADD<=   D00152 D00160	// COLUMN-1 / FEED-X2 INDEX
OUT       M0013F	// FEED X2 LAST INDEX
// ----------------------------------------------------------------------------------
// 
// ----  < 3. TRAY FEEDER X 2 >       SERVO MOTOR STATUS  HOME Search
// 
// ----------------------------------------------------------------------------------
; L51
LOAD      D01040.0	// FEEDER-X2 CtrlReady
AND       D01040.2	// FEEDER-X2 SVD_ON
AND NOT   D01040.6	// FEEDER-X2 SVD BUSY
AND NOT   D01040.A	// FEEDER-X2 Waring
AND NOT   D01040.B	// FEEDER-X2 ModuleErr
AND NOT   D01040.C	// FEEDER-X2 SVD_Err
AND NOT   M0153A	// FEEDER-X2 STOP
AND NOT   M0153F	// FEEDER-X2 MOVE HOLD
OUT       M01530	// FEEDER-X2 READY
; L52
LOAD      M01530	// FEEDER-X2 READY
TON       T0803 1	// FEEDER-X2 READY
; L53
LOAD NOT  M0153F	// FEEDER-X2 MOVE HOLD
AND NOT   M01539	// FEEDER-X2 HOME ->
NOT
TON       T0823 200
// output comment: Motor Not Move °ËÃâ

